Yaskawa INFORM job: u_tourne2TRJ1.JBI

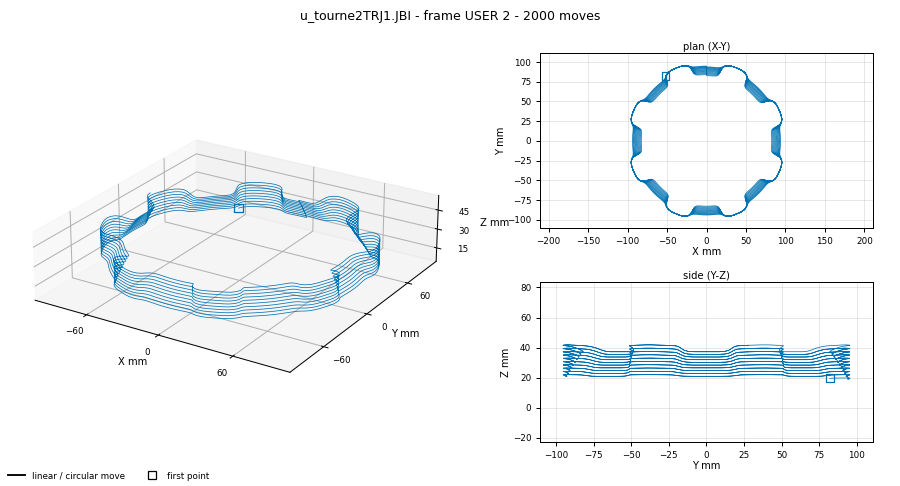
[picture p0: tool path of u_tourne2TRJ1.JBI in frame USER 2, 2000 of 2000 moves have a stored position in this frame; points joined in program order, loops and branches not executed]
/JOB
//NAME u_tourne2TRJ1
///FOLDERNAME DEMO
//POS
///NPOS 2000,0,0,0,0,0
///USER 2
///TOOL 7
///POSTYPE USER
///RECTAN
///RCONF 1,0,0,0,0,0,0,0,0,0,0,0,0,0,0,0,0,0,0,0,0,0,0,0
C00000=-51.961,81.931,19.493,-175.4388,10.0982,0.0000
C00001=-51.163,83.502,19.627,-176.4596,6.1367,0.0000
C00002=-49.917,85.194,19.692,-177.1700,3.1394,0.0000
C00003=-47.874,87.106,19.726,-178.6245,1.1234,0.0000
C00004=-45.272,88.975,19.753,-179.7708,0.1490,0.0000
C00005=-42.449,90.515,19.780,-179.9312,0.0344,0.0000
C00006=-39.659,91.796,19.798,-179.9943,0.0057,0.0000
C00007=-36.867,92.953,19.798,-179.9943,0.0057,0.0000
C00008=-33.988,94.020,19.780,-179.9255,0.0229,0.0000
C00009=-30.903,94.927,19.753,-179.7307,0.0630,0.0000
C00010=-27.741,95.446,19.726,-178.2350,0.1777,0.0000
C00011=-24.945,95.538,19.692,-175.7793,-0.2183,0.0000
C00012=-22.867,95.222,19.627,-173.1679,-1.8469,0.0000
C00013=-21.192,94.676,19.493,-169.6643,-3.9748,0.0000
C00014=-19.540,94.146,19.309,-163.8596,-4.8117,0.0000
C00015=-17.528,93.824,19.120,-157.6161,-2.4729,0.0000
C00016=-14.592,93.857,18.976,-154.0604,1.6120,0.0000
C00017=-10.190,94.262,18.917,-153.0810,2.7315,0.0000
C00018=-5.317,94.652,18.914,-152.9505,1.6728,0.0000
C00019=0.000,94.804,18.916,-152.9225,0.0000,0.0000
C00020=0.000,93.772,20.859,-151.1719,0.0000,0.0000
C00021=5.223,93.624,20.857,-151.1993,-1.7981,0.0000
C00022=10.031,93.243,20.860,-151.3314,-2.8344,0.0000
C00023=14.399,92.874,20.935,-152.4021,-1.1056,0.0000
C00024=17.292,92.935,21.118,-156.8218,4.1655,0.0000
C00025=19.271,93.399,21.361,-164.4290,6.3625,0.0000
C00026=20.902,94.108,21.598,-170.7324,4.7887,0.0000
C00027=22.556,94.852,21.773,-173.9796,2.3281,0.0000
C00028=24.607,95.353,21.858,-176.1467,0.4709,0.0000
C00029=27.423,95.407,21.902,-178.4241,-0.0974,0.0000
C00030=30.651,94.973,21.938,-179.8453,-0.0344,0.0000
C00031=33.828,94.073,21.973,-179.9370,-0.0229,0.0000
C00032=36.813,92.974,21.997,-179.9943,-0.0000,0.0000
C00033=39.712,91.773,21.997,-179.9943,-0.0057,0.0000
C00034=42.599,90.440,21.973,-179.9370,-0.0286,0.0000
C00035=45.483,88.829,21.938,-179.8682,-0.0859,0.0000
C00036=48.072,86.854,21.902,-178.8194,-1.0431,0.0000
C00037=50.025,84.825,21.858,-177.6067,-3.0580,0.0000
C00038=51.121,83.020,21.773,-177.3726,-5.9006,0.0000
C00039=51.765,81.324,21.598,-176.7879,-9.9076,0.0000
C00040=52.416,79.670,21.361,-173.2596,-15.4266,0.0000
C00041=53.488,77.942,21.118,-165.8932,-19.5057,0.0000
C00042=55.491,75.854,20.935,-159.0305,-19.5985,0.0000
C00043=58.840,73.026,20.860,-157.1383,-19.3709,0.0000
C00044=62.509,69.895,20.857,-157.6594,-20.1305,0.0000
C00045=66.307,66.307,20.859,-158.7328,-21.2672,0.0000
C00046=69.895,62.509,20.857,-159.8695,-22.3406,0.0000
C00047=73.026,58.840,20.860,-160.6291,-22.8617,0.0000
C00048=75.854,55.491,20.935,-160.4015,-20.9695,0.0000
C00049=77.942,53.488,21.118,-160.4943,-14.1068,0.0000
C00050=79.670,52.416,21.361,-164.5734,-6.7404,0.0000
C00051=81.324,51.765,21.598,-170.0924,-3.2121,0.0000
C00052=83.020,51.121,21.773,-174.0994,-2.6274,0.0000
C00053=84.825,50.025,21.858,-176.9420,-2.3933,0.0000
C00054=86.854,48.072,21.902,-178.9569,-1.1806,0.0000
C00055=88.829,45.483,21.938,-179.9141,-0.1318,0.0000
C00056=90.440,42.599,21.973,-179.9714,-0.0630,0.0000
C00057=91.773,39.712,21.997,-179.9943,-0.0057,0.0000
C00058=92.974,36.813,21.997,-180.0000,-0.0057,0.0000
C00059=94.073,33.828,21.973,-179.9771,-0.0630,0.0000
C00060=94.973,30.651,21.938,-179.9656,-0.1547,0.0000
C00061=95.407,27.423,21.902,-179.9026,-1.5759,0.0000
C00062=95.353,24.607,21.858,179.5291,-3.8533,0.0000
C00063=94.852,22.556,21.773,177.6719,-6.0204,0.0000
C00064=94.108,20.902,21.598,175.2113,-9.2676,0.0000
C00065=93.399,19.271,21.361,173.6375,-15.5710,0.0000
C00066=92.935,17.292,21.118,175.8345,-23.1782,0.0000
C00067=92.874,14.399,20.935,-178.8944,-27.5979,0.0000
C00068=93.243,10.031,20.860,-177.1656,-28.6686,0.0000
C00069=93.624,5.223,20.857,-178.2019,-28.8007,0.0000
C00070=93.772,0.000,20.859,180.0000,-28.8281,0.0000
C00071=93.624,-5.223,20.857,178.2019,-28.8007,0.0000
C00072=93.243,-10.031,20.860,177.1656,-28.6686,0.0000
C00073=92.875,-14.399,20.935,178.8944,-27.5979,0.0000
C00074=92.935,-17.292,21.118,-175.8345,-23.1782,0.0000
C00075=93.399,-19.271,21.361,-173.6375,-15.5710,0.0000
C00076=94.108,-20.902,21.598,-175.2113,-9.2676,0.0000
C00077=94.852,-22.556,21.773,-177.6719,-6.0204,0.0000
C00078=95.353,-24.607,21.858,-179.5291,-3.8533,0.0000
C00079=95.407,-27.423,21.902,179.9026,-1.5759,0.0000
C00080=94.973,-30.651,21.938,179.9656,-0.1547,0.0000
C00081=94.073,-33.828,21.973,179.9771,-0.0630,0.0000
C00082=92.974,-36.813,21.997,180.0000,-0.0057,0.0000
C00083=91.773,-39.712,21.997,179.9943,-0.0057,0.0000
C00084=90.440,-42.599,21.973,179.9714,-0.0630,0.0000
C00085=88.829,-45.483,21.938,179.9141,-0.1318,0.0000
C00086=86.854,-48.072,21.902,178.9569,-1.1806,0.0000
C00087=84.825,-50.025,21.858,176.9420,-2.3933,0.0000
C00088=83.020,-51.121,21.773,174.0994,-2.6274,0.0000
C00089=81.324,-51.765,21.598,170.0924,-3.2121,0.0000
C00090=79.670,-52.416,21.361,164.5734,-6.7404,0.0000
C00091=77.942,-53.488,21.118,160.4943,-14.1068,0.0000
C00092=75.854,-55.491,20.935,160.4015,-20.9695,0.0000
C00093=73.026,-58.840,20.860,160.6291,-22.8617,0.0000
C00094=69.895,-62.509,20.857,159.8695,-22.3406,0.0000
C00095=66.307,-66.307,20.859,158.7328,-21.2672,0.0000
C00096=62.509,-69.895,20.857,157.6594,-20.1305,0.0000
C00097=58.840,-73.026,20.860,157.1383,-19.3709,0.0000
C00098=55.491,-75.854,20.935,159.0305,-19.5985,0.0000
C00099=53.488,-77.942,21.118,165.8932,-19.5057,0.0000
C00100=52.416,-79.670,21.361,173.2596,-15.4266,0.0000
C00101=51.765,-81.324,21.598,176.7879,-9.9076,0.0000
C00102=51.121,-83.020,21.773,177.3726,-5.9006,0.0000
C00103=50.025,-84.825,21.858,177.6067,-3.0580,0.0000
C00104=48.072,-86.854,21.902,178.8194,-1.0431,0.0000
C00105=45.483,-88.829,21.938,179.8682,-0.0859,0.0000
C00106=42.599,-90.440,21.973,179.9370,-0.0286,0.0000
C00107=39.712,-91.773,21.997,179.9943,-0.0057,0.0000
C00108=36.813,-92.974,21.997,179.9943,-0.0000,0.0000
C00109=33.828,-94.073,21.973,179.9370,-0.0229,0.0000
C00110=30.651,-94.973,21.938,179.8453,-0.0344,0.0000
C00111=27.423,-95.407,21.902,178.4241,-0.0974,0.0000
C00112=24.607,-95.353,21.858,176.1467,0.4709,0.0000
C00113=22.556,-94.852,21.773,173.9796,2.3281,0.0000
C00114=20.902,-94.108,21.598,170.7324,4.7887,0.0000
C00115=19.271,-93.399,21.361,164.4290,6.3625,0.0000
C00116=17.292,-92.935,21.118,156.8218,4.1655,0.0000
C00117=14.399,-92.874,20.935,152.4021,-1.1056,0.0000
C00118=10.031,-93.243,20.860,151.3314,-2.8344,0.0000
C00119=5.223,-93.624,20.857,151.1993,-1.7981,0.0000
C00120=0.000,-93.772,20.859,151.1719,0.0000,0.0000
C00121=0.000,-93.772,20.859,151.1719,0.0000,0.0000
C00122=-5.223,-93.624,20.857,151.1993,1.7981,0.0000
C00123=-10.031,-93.243,20.860,151.3314,2.8344,0.0000
C00124=-14.399,-92.875,20.935,152.4021,1.1056,0.0000
C00125=-17.292,-92.935,21.118,156.8218,-4.1655,0.0000
C00126=-19.271,-93.399,21.361,164.4290,-6.3625,0.0000
C00127=-20.902,-94.108,21.598,170.7324,-4.7887,0.0000
C00128=-22.556,-94.852,21.773,173.9796,-2.3281,0.0000
C00129=-24.607,-95.353,21.858,176.1467,-0.4709,0.0000
C00130=-27.423,-95.407,21.902,178.4241,0.0974,0.0000
C00131=-30.651,-94.973,21.938,179.8453,0.0344,0.0000
C00132=-33.828,-94.073,21.973,179.9370,0.0229,0.0000
C00133=-36.813,-92.974,21.997,179.9943,0.0000,0.0000
C00134=-39.712,-91.773,21.997,179.9943,0.0057,0.0000
C00135=-42.599,-90.440,21.973,179.9370,0.0286,0.0000
C00136=-45.483,-88.829,21.938,179.8682,0.0859,0.0000
C00137=-48.072,-86.854,21.902,178.8194,1.0431,0.0000
C00138=-50.025,-84.825,21.858,177.6067,3.0580,0.0000
C00139=-51.121,-83.020,21.773,177.3726,5.9006,0.0000
C00140=-51.765,-81.324,21.598,176.7879,9.9076,0.0000
C00141=-52.416,-79.670,21.361,173.2596,15.4266,0.0000
C00142=-53.488,-77.942,21.118,165.8932,19.5057,0.0000
C00143=-55.491,-75.854,20.935,159.0305,19.5985,0.0000
C00144=-58.840,-73.026,20.860,157.1383,19.3709,0.0000
C00145=-62.509,-69.895,20.857,157.6594,20.1305,0.0000
C00146=-66.307,-66.307,20.859,158.7328,21.2672,0.0000
C00147=-69.895,-62.509,20.857,159.8695,22.3406,0.0000
C00148=-73.026,-58.840,20.860,160.6291,22.8617,0.0000
C00149=-75.854,-55.491,20.935,160.4015,20.9695,0.0000
C00150=-77.942,-53.488,21.118,160.4943,14.1068,0.0000
C00151=-79.670,-52.416,21.361,164.5734,6.7404,0.0000
C00152=-81.324,-51.765,21.598,170.0924,3.2121,0.0000
C00153=-83.020,-51.121,21.773,174.0994,2.6274,0.0000
C00154=-84.825,-50.025,21.858,176.9420,2.3933,0.0000
C00155=-86.854,-48.072,21.902,178.9569,1.1806,0.0000
C00156=-88.829,-45.483,21.938,179.9141,0.1318,0.0000
C00157=-90.440,-42.599,21.973,179.9714,0.0630,0.0000
C00158=-91.773,-39.712,21.997,179.9943,0.0057,0.0000
C00159=-92.974,-36.813,21.997,180.0000,0.0057,0.0000
C00160=-94.073,-33.828,21.973,179.9771,0.0630,0.0000
C00161=-94.973,-30.651,21.938,179.9656,0.1547,0.0000
C00162=-95.407,-27.423,21.902,179.9026,1.5759,0.0000
C00163=-95.353,-24.607,21.858,-179.5291,3.8533,0.0000
C00164=-94.852,-22.556,21.773,-177.6719,6.0204,0.0000
C00165=-94.108,-20.902,21.598,-175.2113,9.2676,0.0000
C00166=-93.399,-19.271,21.361,-173.6375,15.5710,0.0000
C00167=-92.935,-17.292,21.118,-175.8345,23.1782,0.0000
C00168=-92.874,-14.399,20.935,178.8944,27.5979,0.0000
C00169=-93.243,-10.031,20.860,177.1656,28.6686,0.0000
C00170=-93.624,-5.223,20.857,178.2019,28.8007,0.0000
C00171=-93.772,0.000,20.859,-180.0000,28.8281,0.0000
C00172=-93.624,5.223,20.857,-178.2019,28.8007,0.0000
C00173=-93.243,10.031,20.860,-177.1656,28.6686,0.0000
C00174=-92.875,14.399,20.935,-178.8944,27.5979,0.0000
C00175=-92.935,17.292,21.118,175.8345,23.1782,0.0000
C00176=-93.399,19.271,21.361,173.6375,15.5710,0.0000
C00177=-94.108,20.902,21.598,175.2113,9.2676,0.0000
C00178=-94.852,22.556,21.773,177.6719,6.0204,0.0000
C00179=-95.353,24.607,21.858,179.5291,3.8533,0.0000
C00180=-95.407,27.423,21.902,-179.9026,1.5759,0.0000
C00181=-94.973,30.651,21.938,-179.9656,0.1547,0.0000
C00182=-94.073,33.828,21.973,-179.9771,0.0630,0.0000
C00183=-92.974,36.813,21.997,-180.0000,0.0057,0.0000
C00184=-91.773,39.712,21.997,-179.9943,0.0057,0.0000
C00185=-90.440,42.599,21.973,-179.9714,0.0630,0.0000
C00186=-88.829,45.483,21.938,-179.9141,0.1318,0.0000
C00187=-86.854,48.072,21.902,-178.9569,1.1806,0.0000
C00188=-84.825,50.025,21.858,-176.9420,2.3933,0.0000
C00189=-83.020,51.121,21.773,-174.0994,2.6274,0.0000
C00190=-81.324,51.765,21.598,-170.0924,3.2121,0.0000
C00191=-79.670,52.416,21.361,-164.5734,6.7404,0.0000
C00192=-77.942,53.488,21.118,-160.4943,14.1068,0.0000
C00193=-75.854,55.491,20.935,-160.4015,20.9695,0.0000
C00194=-73.026,58.840,20.860,-160.6291,22.8617,0.0000
C00195=-69.895,62.509,20.857,-159.8695,22.3406,0.0000
C00196=-66.307,66.307,20.859,-158.7328,21.2672,0.0000
C00197=-62.509,69.895,20.857,-157.6594,20.1305,0.0000
C00198=-58.840,73.026,20.860,-157.1383,19.3709,0.0000
C00199=-55.491,75.854,20.935,-159.0305,19.5985,0.0000
C00200=-53.488,77.942,21.118,-165.8932,19.5057,0.0000
C00201=-52.416,79.670,21.361,-173.2596,15.4266,0.0000
C00202=-51.765,81.324,21.598,-176.7879,9.9076,0.0000
C00203=-51.121,83.020,21.773,-177.3726,5.9006,0.0000
C00204=-50.025,84.825,21.858,-177.6067,3.0580,0.0000
C00205=-48.072,86.854,21.902,-178.8194,1.0431,0.0000
C00206=-45.483,88.829,21.938,-179.8682,0.0859,0.0000
C00207=-42.599,90.440,21.973,-179.9370,0.0286,0.0000
C00208=-39.712,91.773,21.997,-179.9943,0.0057,0.0000
C00209=-36.813,92.974,21.997,-179.9943,0.0000,0.0000
C00210=-33.828,94.073,21.973,-179.9370,0.0229,0.0000
C00211=-30.651,94.973,21.938,-179.8453,0.0344,0.0000
C00212=-27.423,95.407,21.902,-178.4241,0.0974,0.0000
C00213=-24.607,95.353,21.858,-176.1467,-0.4709,0.0000
C00214=-22.556,94.852,21.773,-173.9796,-2.3281,0.0000
C00215=-20.902,94.108,21.598,-170.7324,-4.7887,0.0000
C00216=-19.271,93.399,21.361,-164.4290,-6.3625,0.0000
C00217=-17.292,92.935,21.118,-156.8218,-4.1655,0.0000
C00218=-14.399,92.875,20.935,-152.4021,1.1056,0.0000
C00219=-10.031,93.243,20.860,-151.3314,2.8344,0.0000
C00220=-5.223,93.624,20.857,-151.1993,1.7981,0.0000
C00221=0.000,93.772,20.859,-151.1719,0.0000,0.0000
C00222=0.000,92.684,22.771,-149.6091,0.0000,0.0000
C00223=5.124,92.540,22.769,-149.6408,-1.9058,0.0000
C00224=9.864,92.169,22.773,-149.7749,-2.8915,0.0000
C00225=14.194,91.838,22.865,-150.9615,-0.4587,0.0000
C00226=17.042,91.994,23.091,-156.4945,5.9914,0.0000
C00227=18.986,92.606,23.393,-165.5238,7.6283,0.0000
C00228=20.592,93.503,23.691,-172.1229,5.1950,0.0000
C00229=22.223,94.456,23.912,-175.0616,2.5313,0.0000
C00230=24.245,95.156,24.019,-176.7035,0.6543,0.0000
C00231=27.082,95.366,24.075,-178.6935,-0.0287,0.0000
C00232=30.380,95.022,24.120,-179.9771,-0.0057,0.0000
C00233=33.658,94.129,24.166,-179.9427,-0.0172,0.0000
C00234=36.755,92.996,24.196,-179.9943,-0.0000,0.0000
C00235=39.769,91.748,24.196,-179.9943,-0.0000,0.0000
C00236=42.760,90.359,24.166,-179.9484,-0.0229,0.0000
C00237=45.709,88.673,24.120,-179.9828,-0.0115,0.0000
C00238=48.284,86.584,24.075,-179.0544,-0.9055,0.0000
C00239=50.142,84.429,24.019,-178.1296,-2.7928,0.0000
C00240=51.076,82.504,23.912,-178.2908,-5.2754,0.0000
C00241=51.556,80.678,23.691,-178.0785,-9.2060,0.0000
C00242=52.057,78.907,23.393,-174.9767,-15.4952,0.0000
C00243=52.999,77.101,23.091,-166.8652,-20.8965,0.0000
C00244=54.903,74.976,22.865,-158.2902,-21.1534,0.0000
C00245=58.198,72.148,22.773,-155.8794,-20.6200,0.0000
C00246=61.813,69.059,22.769,-156.3563,-21.3360,0.0000
C00247=65.538,65.538,22.771,-157.4774,-22.5226,0.0000
C00248=69.059,61.813,22.769,-158.6640,-23.6437,0.0000
C00249=72.148,58.198,22.773,-159.3800,-24.1206,0.0000
C00250=74.976,54.903,22.865,-158.8466,-21.7155,0.0000
C00251=77.101,52.999,23.091,-159.1035,-13.1348,0.0000
C00252=78.907,52.057,23.393,-164.5048,-5.0233,0.0000
C00253=80.678,51.556,23.691,-170.7940,-1.9215,0.0000
C00254=82.504,51.076,23.912,-174.7246,-1.7092,0.0000
C00255=84.429,50.142,24.019,-177.2072,-1.8704,0.0000
C00256=86.584,48.284,24.075,-179.0945,-0.9456,0.0000
C00257=88.673,45.709,24.120,-179.9885,-0.0172,0.0000
C00258=90.359,42.760,24.166,-179.9771,-0.0516,0.0000
C00259=91.748,39.769,24.196,-180.0000,-0.0057,0.0000
C00260=92.996,36.755,24.196,-180.0000,-0.0057,0.0000
C00261=94.129,33.658,24.166,-179.9828,-0.0573,0.0000
C00262=95.022,30.380,24.120,-179.9943,-0.0229,0.0000
C00263=95.366,27.082,24.075,-179.9713,-1.3065,0.0000
C00264=95.156,24.245,24.019,179.3457,-3.2965,0.0000
C00265=94.456,22.223,23.912,177.4687,-4.9384,0.0000
C00266=93.503,20.592,23.691,174.8050,-7.8771,0.0000
C00267=92.606,18.986,23.393,172.3717,-14.4762,0.0000
C00268=91.994,17.042,23.091,174.0086,-23.5055,0.0000
C00269=91.838,14.194,22.865,-179.5413,-29.0385,0.0000
C00270=92.169,9.864,22.773,-177.1085,-30.2251,0.0000
C00271=92.540,5.124,22.769,-178.0942,-30.3592,0.0000
C00272=92.684,0.000,22.771,180.0000,-30.3909,0.0000
C00273=92.540,-5.124,22.769,178.0942,-30.3592,0.0000
C00274=92.169,-9.864,22.773,177.1085,-30.2251,0.0000
C00275=91.838,-14.194,22.865,179.5413,-29.0385,0.0000
C00276=91.994,-17.042,23.091,-174.0086,-23.5055,0.0000
C00277=92.606,-18.986,23.393,-172.3717,-14.4762,0.0000
C00278=93.503,-20.592,23.691,-174.8050,-7.8771,0.0000
C00279=94.456,-22.223,23.912,-177.4687,-4.9384,0.0000
C00280=95.156,-24.245,24.019,-179.3457,-3.2965,0.0000
C00281=95.366,-27.082,24.075,179.9713,-1.3065,0.0000
C00282=95.022,-30.380,24.120,179.9943,-0.0229,0.0000
C00283=94.129,-33.658,24.166,179.9828,-0.0573,0.0000
C00284=92.996,-36.755,24.196,180.0000,-0.0057,0.0000
C00285=91.748,-39.769,24.196,180.0000,-0.0057,0.0000
C00286=90.359,-42.760,24.166,179.9771,-0.0516,0.0000
C00287=88.673,-45.709,24.120,179.9885,-0.0172,0.0000
C00288=86.584,-48.284,24.075,179.0945,-0.9456,0.0000
C00289=84.429,-50.142,24.019,177.2072,-1.8704,0.0000
C00290=82.504,-51.076,23.912,174.7246,-1.7092,0.0000
C00291=80.678,-51.556,23.691,170.7940,-1.9215,0.0000
C00292=78.907,-52.057,23.393,164.5048,-5.0233,0.0000
C00293=77.101,-52.999,23.091,159.1035,-13.1348,0.0000
C00294=74.976,-54.903,22.865,158.8466,-21.7098,0.0000
C00295=72.148,-58.198,22.773,159.3800,-24.1206,0.0000
C00296=69.059,-61.813,22.769,158.6640,-23.6437,0.0000
C00297=65.538,-65.538,22.771,157.4774,-22.5226,0.0000
C00298=61.813,-69.059,22.769,156.3563,-21.3360,0.0000
C00299=58.198,-72.148,22.773,155.8794,-20.6200,0.0000
C00300=54.903,-74.976,22.865,158.2845,-21.1534,0.0000
C00301=52.999,-77.101,23.091,166.8652,-20.8965,0.0000
C00302=52.057,-78.907,23.393,174.9767,-15.4952,0.0000
C00303=51.556,-80.678,23.691,178.0785,-9.2060,0.0000
C00304=51.076,-82.504,23.912,178.2908,-5.2754,0.0000
C00305=50.142,-84.429,24.019,178.1296,-2.7928,0.0000
C00306=48.284,-86.584,24.075,179.0544,-0.9055,0.0000
C00307=45.709,-88.673,24.120,179.9828,-0.0115,0.0000
C00308=42.760,-90.359,24.166,179.9484,-0.0229,0.0000
C00309=39.769,-91.748,24.196,179.9943,-0.0000,0.0000
C00310=36.755,-92.996,24.196,179.9943,-0.0000,0.0000
C00311=33.658,-94.129,24.166,179.9427,-0.0172,0.0000
C00312=30.380,-95.022,24.120,179.9771,-0.0057,0.0000
C00313=27.082,-95.366,24.075,178.6935,-0.0287,0.0000
C00314=24.245,-95.156,24.019,176.7035,0.6543,0.0000
C00315=22.223,-94.456,23.912,175.0616,2.5313,0.0000
C00316=20.592,-93.503,23.691,172.1229,5.1950,0.0000
C00317=18.986,-92.606,23.393,165.5238,7.6283,0.0000
C00318=17.042,-91.994,23.091,156.4945,5.9914,0.0000
C00319=14.194,-91.838,22.865,150.9615,-0.4587,0.0000
C00320=9.864,-92.169,22.773,149.7749,-2.8915,0.0000
C00321=5.124,-92.540,22.769,149.6408,-1.9058,0.0000
C00322=0.000,-92.684,22.771,149.6091,0.0000,0.0000
C00323=0.000,-92.684,22.771,149.6091,0.0000,0.0000
C00324=-5.124,-92.540,22.769,149.6408,1.9058,0.0000
C00325=-9.864,-92.169,22.773,149.7749,2.8915,0.0000
C00326=-14.194,-91.838,22.865,150.9615,0.4587,0.0000
C00327=-17.042,-91.994,23.091,156.4945,-5.9914,0.0000
C00328=-18.986,-92.606,23.393,165.5238,-7.6283,0.0000
C00329=-20.592,-93.503,23.691,172.1229,-5.1950,0.0000
C00330=-22.223,-94.456,23.912,175.0616,-2.5313,0.0000
C00331=-24.245,-95.156,24.019,176.7035,-0.6543,0.0000
C00332=-27.082,-95.366,24.075,178.6935,0.0287,0.0000
C00333=-30.380,-95.022,24.120,179.9771,0.0057,0.0000
C00334=-33.658,-94.129,24.166,179.9427,0.0172,0.0000
C00335=-36.755,-92.996,24.196,179.9943,0.0000,0.0000
C00336=-39.769,-91.748,24.196,179.9943,0.0000,0.0000
C00337=-42.760,-90.359,24.166,179.9484,0.0229,0.0000
C00338=-45.709,-88.673,24.120,179.9828,0.0115,0.0000
C00339=-48.284,-86.584,24.075,179.0544,0.9055,0.0000
C00340=-50.142,-84.429,24.019,178.1296,2.7928,0.0000
C00341=-51.076,-82.504,23.912,178.2908,5.2754,0.0000
C00342=-51.556,-80.678,23.691,178.0785,9.2060,0.0000
C00343=-52.057,-78.907,23.393,174.9767,15.4952,0.0000
C00344=-52.999,-77.101,23.091,166.8652,20.8965,0.0000
C00345=-54.903,-74.976,22.865,158.2902,21.1534,0.0000
C00346=-58.198,-72.148,22.773,155.8794,20.6200,0.0000
C00347=-61.813,-69.059,22.769,156.3563,21.3360,0.0000
C00348=-65.538,-65.538,22.771,157.4774,22.5226,0.0000
C00349=-69.059,-61.813,22.769,158.6640,23.6437,0.0000
C00350=-72.148,-58.198,22.773,159.3800,24.1206,0.0000
C00351=-74.976,-54.903,22.865,158.8466,21.7155,0.0000
C00352=-77.101,-52.999,23.091,159.1035,13.1348,0.0000
C00353=-78.907,-52.057,23.393,164.5048,5.0233,0.0000
C00354=-80.678,-51.556,23.691,170.7940,1.9215,0.0000
C00355=-82.504,-51.076,23.912,174.7246,1.7092,0.0000
C00356=-84.429,-50.142,24.019,177.2072,1.8704,0.0000
C00357=-86.584,-48.284,24.075,179.0945,0.9456,0.0000
C00358=-88.673,-45.709,24.120,179.9885,0.0172,0.0000
C00359=-90.359,-42.760,24.166,179.9771,0.0516,0.0000
C00360=-91.748,-39.769,24.196,180.0000,0.0057,0.0000
C00361=-92.996,-36.755,24.196,180.0000,0.0057,0.0000
C00362=-94.129,-33.658,24.166,179.9828,0.0573,0.0000
C00363=-95.022,-30.380,24.120,179.9943,0.0229,0.0000
C00364=-95.366,-27.082,24.075,179.9713,1.3065,0.0000
C00365=-95.156,-24.245,24.019,-179.3457,3.2965,0.0000
C00366=-94.456,-22.223,23.912,-177.4687,4.9384,0.0000
C00367=-93.503,-20.592,23.691,-174.8050,7.8771,0.0000
C00368=-92.606,-18.986,23.393,-172.3717,14.4762,0.0000
C00369=-91.994,-17.042,23.091,-174.0086,23.5055,0.0000
C00370=-91.838,-14.194,22.865,179.5413,29.0385,0.0000
C00371=-92.169,-9.864,22.773,177.1085,30.2251,0.0000
C00372=-92.540,-5.124,22.769,178.0942,30.3592,0.0000
C00373=-92.684,0.000,22.771,-180.0000,30.3909,0.0000
C00374=-92.540,5.124,22.769,-178.0942,30.3592,0.0000
C00375=-92.169,9.864,22.773,-177.1085,30.2251,0.0000
C00376=-91.838,14.194,22.865,-179.5413,29.0385,0.0000
C00377=-91.994,17.042,23.091,174.0086,23.5055,0.0000
C00378=-92.606,18.986,23.393,172.3717,14.4762,0.0000
C00379=-93.503,20.592,23.691,174.8050,7.8771,0.0000
C00380=-94.456,22.223,23.912,177.4687,4.9384,0.0000
C00381=-95.156,24.245,24.019,179.3457,3.2965,0.0000
C00382=-95.366,27.082,24.075,-179.9713,1.3065,0.0000
C00383=-95.022,30.380,24.120,-179.9943,0.0229,0.0000
C00384=-94.129,33.658,24.166,-179.9828,0.0573,0.0000
C00385=-92.996,36.755,24.196,-180.0000,0.0057,0.0000
C00386=-91.748,39.769,24.196,-180.0000,0.0057,0.0000
C00387=-90.359,42.760,24.166,-179.9771,0.0516,0.0000
C00388=-88.673,45.709,24.120,-179.9885,0.0172,0.0000
C00389=-86.584,48.284,24.075,-179.0945,0.9456,0.0000
C00390=-84.429,50.142,24.019,-177.2072,1.8704,0.0000
C00391=-82.504,51.076,23.912,-174.7246,1.7092,0.0000
C00392=-80.678,51.556,23.691,-170.7940,1.9215,0.0000
C00393=-78.907,52.057,23.393,-164.5048,5.0233,0.0000
C00394=-77.101,52.999,23.091,-159.1035,13.1348,0.0000
C00395=-74.976,54.903,22.865,-158.8466,21.7098,0.0000
C00396=-72.148,58.198,22.773,-159.3800,24.1206,0.0000
C00397=-69.059,61.813,22.769,-158.6640,23.6437,0.0000
C00398=-65.538,65.538,22.771,-157.4774,22.5226,0.0000
C00399=-61.813,69.059,22.769,-156.3563,21.3360,0.0000
C00400=-58.198,72.148,22.773,-155.8794,20.6200,0.0000
C00401=-54.903,74.976,22.865,-158.2845,21.1534,0.0000
C00402=-52.999,77.101,23.091,-166.8652,20.8965,0.0000
C00403=-52.057,78.907,23.393,-174.9767,15.4952,0.0000
C00404=-51.556,80.678,23.691,-178.0785,9.2060,0.0000
C00405=-51.076,82.504,23.912,-178.2908,5.2754,0.0000
C00406=-50.142,84.429,24.019,-178.1296,2.7928,0.0000
C00407=-48.284,86.584,24.075,-179.0544,0.9055,0.0000
C00408=-45.709,88.673,24.120,-179.9828,0.0115,0.0000
C00409=-42.760,90.359,24.166,-179.9484,0.0229,0.0000
C00410=-39.769,91.748,24.196,-179.9943,0.0000,0.0000
C00411=-36.755,92.996,24.196,-179.9943,0.0000,0.0000
C00412=-33.658,94.129,24.166,-179.9427,0.0172,0.0000
C00413=-30.380,95.022,24.120,-179.9771,0.0057,0.0000
C00414=-27.082,95.366,24.075,-178.6935,0.0287,0.0000
C00415=-24.245,95.156,24.019,-176.7035,-0.6543,0.0000
C00416=-22.223,94.456,23.912,-175.0616,-2.5313,0.0000
C00417=-20.592,93.503,23.691,-172.1229,-5.1950,0.0000
C00418=-18.986,92.606,23.393,-165.5238,-7.6283,0.0000
C00419=-17.042,91.994,23.091,-156.4945,-5.9914,0.0000
C00420=-14.194,91.838,22.865,-150.9615,0.4587,0.0000
C00421=-9.864,92.169,22.773,-149.7749,2.8915,0.0000
C00422=-5.124,92.540,22.769,-149.6408,1.9058,0.0000
C00423=0.000,92.684,22.771,-149.6091,0.0000,0.0000
C00424=0.000,91.548,24.655,-148.2236,0.0000,0.0000
C00425=5.020,91.408,24.652,-148.2498,-2.0079,0.0000
C00426=9.690,91.047,24.657,-148.3861,-2.9135,0.0000
C00427=13.981,90.755,24.767,-149.7221,0.3185,0.0000
C00428=16.781,91.008,25.041,-156.6444,7.8331,0.0000
C00429=18.686,91.772,25.406,-167.0184,8.4700,0.0000
C00430=20.265,92.865,25.771,-173.6420,5.1605,0.0000
C00431=21.871,94.037,26.043,-176.2870,2.4065,0.0000
C00432=23.861,94.948,26.175,-177.4320,0.7169,0.0000
C00433=26.720,95.323,26.245,-179.0317,0.0229,0.0000
C00434=30.093,95.074,26.301,179.8682,0.0229,0.0000
C00435=33.476,94.189,26.358,-179.9599,-0.0172,0.0000
C00436=36.693,93.020,26.395,-179.9943,-0.0000,0.0000
C00437=39.829,91.721,26.395,-179.9943,-0.0000,0.0000
C00438=42.931,90.273,26.358,-179.9599,-0.0172,0.0000
C00439=45.948,88.507,26.301,179.8911,0.0802,0.0000
C00440=48.509,86.297,26.245,-179.3296,-0.6990,0.0000
C00441=50.266,84.010,26.175,-178.6924,-2.3275,0.0000
C00442=51.029,81.959,26.043,-179.0748,-4.3249,0.0000
C00443=51.336,79.995,25.771,-179.1434,-8.1179,0.0000
C00444=51.679,78.105,25.406,-176.7001,-15.0175,0.0000
C00445=52.487,76.218,25.041,-168.2468,-21.9304,0.0000
C00446=54.287,74.059,24.767,-157.7618,-22.6236,0.0000
C00447=57.528,71.231,24.657,-154.7700,-21.7654,0.0000
C00448=61.085,68.184,24.652,-155.1864,-22.4262,0.0000
C00449=64.734,64.734,24.655,-156.3434,-23.6566,0.0000
C00450=68.184,61.085,24.652,-157.5738,-24.8136,0.0000
C00451=71.231,57.528,24.657,-158.2346,-25.2300,0.0000
C00452=74.059,54.287,24.767,-157.3764,-22.2382,0.0000
C00453=76.218,52.487,25.041,-158.0696,-11.7532,0.0000
C00454=78.105,51.679,25.406,-164.9825,-3.2999,0.0000
C00455=79.995,51.336,25.771,-171.8821,-0.8566,0.0000
C00456=81.959,51.029,26.043,-175.6751,-0.9252,0.0000
C00457=84.010,50.266,26.175,-177.6725,-1.3076,0.0000
C00458=86.297,48.509,26.245,-179.3010,-0.6704,0.0000
C00459=88.507,45.948,26.301,179.9198,0.1089,0.0000
C00460=90.273,42.931,26.358,-179.9828,-0.0401,0.0000
C00461=91.721,39.829,26.395,-180.0000,-0.0057,0.0000
C00462=93.020,36.693,26.395,-180.0000,-0.0057,0.0000
C00463=94.189,33.476,26.358,-179.9828,-0.0401,0.0000
C00464=95.074,30.093,26.301,179.9771,0.1318,0.0000
C00465=95.323,26.720,26.245,179.9771,-0.9683,0.0000
C00466=94.948,23.861,26.175,179.2831,-2.5680,0.0000
C00467=94.037,21.871,26.043,177.5935,-3.7130,0.0000
C00468=92.865,20.265,25.771,174.8395,-6.3580,0.0000
C00469=91.772,18.686,25.406,171.5300,-12.9816,0.0000
C00470=91.008,16.781,25.041,172.1669,-23.3556,0.0000
C00471=90.755,13.981,24.767,179.6815,-30.2779,0.0000
C00472=91.047,9.690,24.657,-177.0865,-31.6139,0.0000
C00473=91.408,5.020,24.652,-177.9921,-31.7502,0.0000
C00474=91.548,0.000,24.655,180.0000,-31.7764,0.0000
C00475=91.408,-5.020,24.652,177.9921,-31.7502,0.0000
C00476=91.047,-9.690,24.657,177.0865,-31.6139,0.0000
C00477=90.755,-13.981,24.767,-179.6815,-30.2779,0.0000
C00478=91.008,-16.781,25.041,-172.1669,-23.3556,0.0000
C00479=91.772,-18.686,25.406,-171.5300,-12.9816,0.0000
C00480=92.865,-20.265,25.771,-174.8395,-6.3580,0.0000
C00481=94.037,-21.871,26.043,-177.5935,-3.7130,0.0000
C00482=94.948,-23.861,26.175,-179.2831,-2.5680,0.0000
C00483=95.323,-26.720,26.245,-179.9771,-0.9683,0.0000
C00484=95.074,-30.093,26.301,-179.9771,0.1318,0.0000
C00485=94.189,-33.476,26.358,179.9828,-0.0401,0.0000
C00486=93.020,-36.693,26.395,180.0000,-0.0057,0.0000
C00487=91.721,-39.829,26.395,180.0000,-0.0057,0.0000
C00488=90.273,-42.931,26.358,179.9828,-0.0401,0.0000
C00489=88.507,-45.948,26.301,-179.9198,0.1089,0.0000
C00490=86.297,-48.509,26.245,179.3010,-0.6704,0.0000
C00491=84.010,-50.266,26.175,177.6725,-1.3076,0.0000
C00492=81.959,-51.029,26.043,175.6751,-0.9252,0.0000
C00493=79.995,-51.336,25.771,171.8821,-0.8566,0.0000
C00494=78.105,-51.679,25.406,164.9825,-3.2999,0.0000
C00495=76.218,-52.487,25.041,158.0696,-11.7532,0.0000
C00496=74.059,-54.287,24.767,157.3764,-22.2382,0.0000
C00497=71.231,-57.528,24.657,158.2346,-25.2300,0.0000
C00498=68.184,-61.085,24.652,157.5738,-24.8136,0.0000
C00499=64.734,-64.734,24.655,156.3434,-23.6566,0.0000
C00500=61.085,-68.184,24.652,155.1864,-22.4262,0.0000
C00501=57.528,-71.231,24.657,154.7700,-21.7654,0.0000
C00502=54.287,-74.059,24.767,157.7618,-22.6236,0.0000
C00503=52.487,-76.218,25.041,168.2468,-21.9304,0.0000
C00504=51.679,-78.105,25.406,176.7001,-15.0175,0.0000
C00505=51.336,-79.995,25.771,179.1434,-8.1179,0.0000
C00506=51.029,-81.959,26.043,179.0748,-4.3249,0.0000
C00507=50.266,-84.010,26.175,178.6924,-2.3275,0.0000
C00508=48.509,-86.297,26.245,179.3296,-0.6990,0.0000
C00509=45.948,-88.507,26.301,-179.8911,0.0802,0.0000
C00510=42.931,-90.273,26.358,179.9599,-0.0172,0.0000
C00511=39.829,-91.721,26.395,179.9943,-0.0000,0.0000
C00512=36.693,-93.020,26.395,179.9943,-0.0000,0.0000
C00513=33.476,-94.189,26.358,179.9599,-0.0172,0.0000
C00514=30.093,-95.074,26.301,-179.8682,0.0229,0.0000
C00515=26.720,-95.323,26.245,179.0317,0.0229,0.0000
C00516=23.861,-94.948,26.175,177.4320,0.7169,0.0000
C00517=21.871,-94.037,26.043,176.2870,2.4065,0.0000
C00518=20.265,-92.865,25.771,173.6420,5.1605,0.0000
C00519=18.686,-91.772,25.406,167.0184,8.4700,0.0000
C00520=16.781,-91.008,25.041,156.6444,7.8331,0.0000
C00521=13.981,-90.755,24.767,149.7221,0.3185,0.0000
C00522=9.690,-91.047,24.657,148.3861,-2.9135,0.0000
C00523=5.020,-91.408,24.652,148.2498,-2.0079,0.0000
C00524=0.000,-91.548,24.655,148.2236,0.0000,0.0000
C00525=0.000,-91.548,24.655,148.2236,0.0000,0.0000
C00526=-5.020,-91.408,24.652,148.2498,2.0079,0.0000
C00527=-9.690,-91.047,24.657,148.3861,2.9135,0.0000
C00528=-13.981,-90.755,24.767,149.7221,-0.3185,0.0000
C00529=-16.781,-91.008,25.041,156.6444,-7.8331,0.0000
C00530=-18.686,-91.772,25.406,167.0184,-8.4700,0.0000
C00531=-20.265,-92.865,25.771,173.6420,-5.1605,0.0000
C00532=-21.871,-94.037,26.043,176.2870,-2.4065,0.0000
C00533=-23.861,-94.948,26.175,177.4320,-0.7169,0.0000
C00534=-26.720,-95.323,26.245,179.0317,-0.0229,0.0000
C00535=-30.093,-95.074,26.301,-179.8682,-0.0229,0.0000
C00536=-33.476,-94.189,26.358,179.9599,0.0172,0.0000
C00537=-36.693,-93.020,26.395,179.9943,0.0000,0.0000
C00538=-39.829,-91.721,26.395,179.9943,0.0000,0.0000
C00539=-42.931,-90.273,26.358,179.9599,0.0172,0.0000
C00540=-45.948,-88.507,26.301,-179.8911,-0.0802,0.0000
C00541=-48.509,-86.297,26.245,179.3296,0.6990,0.0000
C00542=-50.266,-84.010,26.175,178.6924,2.3275,0.0000
C00543=-51.029,-81.959,26.043,179.0748,4.3249,0.0000
C00544=-51.336,-79.995,25.771,179.1434,8.1179,0.0000
C00545=-51.679,-78.105,25.406,176.7001,15.0175,0.0000
C00546=-52.487,-76.218,25.041,168.2468,21.9304,0.0000
C00547=-54.287,-74.059,24.767,157.7618,22.6236,0.0000
C00548=-57.528,-71.231,24.657,154.7700,21.7654,0.0000
C00549=-61.085,-68.184,24.652,155.1864,22.4262,0.0000
C00550=-64.734,-64.734,24.655,156.3434,23.6566,0.0000
C00551=-68.184,-61.085,24.652,157.5738,24.8136,0.0000
C00552=-71.231,-57.528,24.657,158.2346,25.2300,0.0000
C00553=-74.059,-54.287,24.767,157.3764,22.2382,0.0000
C00554=-76.218,-52.487,25.041,158.0696,11.7532,0.0000
C00555=-78.105,-51.679,25.406,164.9825,3.2999,0.0000
C00556=-79.995,-51.336,25.771,171.8821,0.8566,0.0000
C00557=-81.959,-51.029,26.043,175.6751,0.9252,0.0000
C00558=-84.010,-50.266,26.175,177.6725,1.3076,0.0000
C00559=-86.297,-48.509,26.245,179.3010,0.6704,0.0000
C00560=-88.507,-45.948,26.301,-179.9198,-0.1089,0.0000
C00561=-90.273,-42.931,26.358,179.9828,0.0401,0.0000
C00562=-91.721,-39.829,26.395,180.0000,0.0057,0.0000
C00563=-93.020,-36.693,26.395,180.0000,0.0057,0.0000
C00564=-94.189,-33.476,26.358,179.9828,0.0401,0.0000
C00565=-95.074,-30.093,26.301,-179.9771,-0.1318,0.0000
C00566=-95.323,-26.720,26.245,-179.9771,0.9683,0.0000
C00567=-94.948,-23.861,26.175,-179.2831,2.5680,0.0000
C00568=-94.037,-21.871,26.043,-177.5935,3.7130,0.0000
C00569=-92.865,-20.265,25.771,-174.8395,6.3580,0.0000
C00570=-91.772,-18.686,25.406,-171.5300,12.9816,0.0000
C00571=-91.008,-16.781,25.041,-172.1669,23.3556,0.0000
C00572=-90.755,-13.981,24.767,-179.6815,30.2779,0.0000
C00573=-91.047,-9.690,24.657,177.0865,31.6139,0.0000
C00574=-91.408,-5.020,24.652,177.9921,31.7502,0.0000
C00575=-91.548,0.000,24.655,-180.0000,31.7764,0.0000
C00576=-91.408,5.020,24.652,-177.9921,31.7502,0.0000
C00577=-91.047,9.690,24.657,-177.0865,31.6139,0.0000
C00578=-90.755,13.981,24.767,179.6815,30.2779,0.0000
C00579=-91.008,16.781,25.041,172.1669,23.3556,0.0000
C00580=-91.772,18.686,25.406,171.5300,12.9816,0.0000
C00581=-92.865,20.265,25.771,174.8395,6.3580,0.0000
C00582=-94.037,21.871,26.043,177.5935,3.7130,0.0000
C00583=-94.948,23.861,26.175,179.2831,2.5680,0.0000
C00584=-95.323,26.720,26.245,179.9771,0.9683,0.0000
C00585=-95.074,30.093,26.301,179.9771,-0.1318,0.0000
C00586=-94.189,33.476,26.358,-179.9828,0.0401,0.0000
C00587=-93.020,36.693,26.395,-180.0000,0.0057,0.0000
C00588=-91.721,39.829,26.395,-180.0000,0.0057,0.0000
C00589=-90.273,42.931,26.358,-179.9828,0.0401,0.0000
C00590=-88.507,45.948,26.301,179.9198,-0.1089,0.0000
C00591=-86.297,48.509,26.245,-179.3010,0.6704,0.0000
C00592=-84.010,50.266,26.175,-177.6725,1.3076,0.0000
C00593=-81.959,51.029,26.043,-175.6751,0.9252,0.0000
C00594=-79.995,51.336,25.771,-171.8821,0.8566,0.0000
C00595=-78.105,51.679,25.406,-164.9825,3.2999,0.0000
C00596=-76.218,52.487,25.041,-158.0696,11.7532,0.0000
C00597=-74.059,54.287,24.767,-157.3764,22.2382,0.0000
C00598=-71.231,57.528,24.657,-158.2346,25.2300,0.0000
C00599=-68.184,61.085,24.652,-157.5738,24.8136,0.0000
C00600=-64.734,64.734,24.655,-156.3434,23.6566,0.0000
C00601=-61.085,68.184,24.652,-155.1864,22.4262,0.0000
C00602=-57.528,71.231,24.657,-154.7700,21.7654,0.0000
C00603=-54.287,74.059,24.767,-157.7618,22.6236,0.0000
C00604=-52.487,76.218,25.041,-168.2468,21.9304,0.0000
C00605=-51.679,78.105,25.406,-176.7001,15.0175,0.0000
C00606=-51.336,79.995,25.771,-179.1434,8.1179,0.0000
C00607=-51.029,81.959,26.043,-179.0748,4.3249,0.0000
C00608=-50.266,84.010,26.175,-178.6924,2.3275,0.0000
C00609=-48.509,86.297,26.245,-179.3296,0.6990,0.0000
C00610=-45.948,88.507,26.301,179.8911,-0.0802,0.0000
C00611=-42.931,90.273,26.358,-179.9599,0.0172,0.0000
C00612=-39.829,91.721,26.395,-179.9943,0.0000,0.0000
C00613=-36.693,93.020,26.395,-179.9943,0.0000,0.0000
C00614=-33.476,94.189,26.358,-179.9599,0.0172,0.0000
C00615=-30.093,95.074,26.301,179.8682,-0.0229,0.0000
C00616=-26.720,95.323,26.245,-179.0317,-0.0229,0.0000
C00617=-23.861,94.948,26.175,-177.4320,-0.7169,0.0000
C00618=-21.871,94.037,26.043,-176.2870,-2.4065,0.0000
C00619=-20.265,92.865,25.771,-173.6420,-5.1605,0.0000
C00620=-18.686,91.772,25.406,-167.0184,-8.4700,0.0000
C00621=-16.781,91.008,25.041,-156.6444,-7.8331,0.0000
C00622=-13.981,90.755,24.767,-149.7221,-0.3185,0.0000
C00623=-9.690,91.047,24.657,-148.3861,2.9135,0.0000
C00624=-5.020,91.408,24.652,-148.2498,2.0079,0.0000
C00625=0.000,91.548,24.655,-148.2236,0.0000,0.0000
C00626=0.000,90.369,26.513,-146.9901,0.0000,0.0000
C00627=4.912,90.233,26.509,-147.0206,-2.0968,0.0000
C00628=9.508,89.882,26.515,-147.1593,-2.8985,0.0000
C00629=13.759,89.629,26.645,-148.6805,1.2140,0.0000
C00630=16.509,89.983,26.968,-157.2651,9.5602,0.0000
C00631=18.373,90.901,27.402,-168.7355,8.8469,0.0000
C00632=19.923,92.196,27.838,-175.1304,4.7436,0.0000
C00633=21.502,93.597,28.166,-177.5226,1.9674,0.0000
C00634=23.458,94.728,28.327,-178.2693,0.6305,0.0000
C00635=26.340,95.277,28.411,-179.4213,0.0344,0.0000
C00636=29.791,95.129,28.479,179.6963,0.0458,0.0000
C00637=33.285,94.252,28.548,-179.9714,-0.0115,0.0000
C00638=36.628,93.045,28.594,-180.0000,-0.0000,0.0000
C00639=39.893,91.693,28.594,-180.0000,-0.0000,0.0000
C00640=43.110,90.182,28.548,-179.9714,-0.0115,0.0000
C00641=46.201,88.332,28.479,179.7536,0.1833,0.0000
C00642=48.746,85.996,28.411,-179.6161,-0.4355,0.0000
C00643=50.396,83.570,28.327,-179.2262,-1.6677,0.0000
C00644=50.979,81.387,28.166,-179.6385,-3.1414,0.0000
C00645=51.105,79.281,27.838,-179.9077,-6.7825,0.0000
C00646=51.285,77.269,27.402,-178.2394,-14.0877,0.0000
C00647=51.954,75.301,26.968,-169.9515,-22.5582,0.0000
C00648=53.649,73.106,26.645,-157.4473,-24.0017,0.0000
C00649=56.833,70.280,26.515,-153.7965,-22.8144,0.0000
C00650=60.331,67.277,26.509,-154.1417,-23.4086,0.0000
C00651=63.901,63.901,26.513,-155.3289,-24.6711,0.0000
C00652=67.277,60.331,26.509,-156.5914,-25.8583,0.0000
C00653=70.280,56.833,26.515,-157.1856,-26.2035,0.0000
C00654=73.106,53.649,26.645,-155.9983,-22.5527,0.0000
C00655=75.301,51.954,26.968,-157.4418,-10.0485,0.0000
C00656=77.269,51.285,27.402,-165.9123,-1.7606,0.0000
C00657=79.281,51.105,27.838,-173.2175,-0.0923,0.0000
C00658=81.387,50.979,28.166,-176.8586,-0.3615,0.0000
C00659=83.570,50.396,28.327,-178.3323,-0.7738,0.0000
C00660=85.996,48.746,28.411,-179.5645,-0.3839,0.0000
C00661=88.332,46.201,28.479,179.8167,0.2464,0.0000
C00662=90.182,43.110,28.548,-179.9885,-0.0286,0.0000
C00663=91.693,39.893,28.594,-180.0000,-0.0000,0.0000
C00664=93.045,36.628,28.594,-180.0000,-0.0000,0.0000
C00665=94.252,33.285,28.548,-179.9885,-0.0286,0.0000
C00666=95.129,29.791,28.479,179.9542,0.3037,0.0000
C00667=95.277,26.340,28.411,179.9656,-0.5787,0.0000
C00668=94.728,23.458,28.327,179.3695,-1.7307,0.0000
C00669=93.597,21.502,28.166,178.0326,-2.4774,0.0000
C00670=92.196,19.923,27.838,175.2564,-4.8696,0.0000
C00671=90.901,18.373,27.402,171.1531,-11.2645,0.0000
C00672=89.983,16.509,26.968,170.4398,-22.7349,0.0000
C00673=89.629,13.759,26.645,178.7860,-31.3195,0.0000
C00674=89.882,9.508,26.515,-177.1015,-32.8407,0.0000
C00675=90.233,4.912,26.509,-177.9032,-32.9794,0.0000
C00676=90.369,0.000,26.513,180.0000,-33.0099,0.0000
C00677=90.233,-4.912,26.509,177.9032,-32.9794,0.0000
C00678=89.882,-9.508,26.515,177.1015,-32.8407,0.0000
C00679=89.629,-13.759,26.645,-178.7860,-31.3195,0.0000
C00680=89.983,-16.509,26.968,-170.4398,-22.7349,0.0000
C00681=90.901,-18.373,27.402,-171.1531,-11.2645,0.0000
C00682=92.196,-19.923,27.838,-175.2564,-4.8696,0.0000
C00683=93.597,-21.502,28.166,-178.0326,-2.4774,0.0000
C00684=94.728,-23.458,28.327,-179.3695,-1.7307,0.0000
C00685=95.277,-26.340,28.411,-179.9656,-0.5787,0.0000
C00686=95.129,-29.791,28.479,-179.9542,0.3037,0.0000
C00687=94.252,-33.285,28.548,179.9885,-0.0286,0.0000
C00688=93.045,-36.628,28.594,180.0000,-0.0000,0.0000
C00689=91.693,-39.893,28.594,180.0000,-0.0000,0.0000
C00690=90.182,-43.110,28.548,179.9885,-0.0286,0.0000
C00691=88.332,-46.201,28.479,-179.8167,0.2464,0.0000
C00692=85.996,-48.746,28.411,179.5645,-0.3839,0.0000
C00693=83.570,-50.396,28.327,178.3323,-0.7738,0.0000
C00694=81.387,-50.979,28.166,176.8586,-0.3615,0.0000
C00695=79.281,-51.105,27.838,173.2175,-0.0923,0.0000
C00696=77.269,-51.285,27.402,165.9123,-1.7606,0.0000
C00697=75.301,-51.954,26.968,157.4418,-10.0485,0.0000
C00698=73.106,-53.649,26.645,155.9983,-22.5527,0.0000
C00699=70.280,-56.833,26.515,157.1856,-26.2035,0.0000
C00700=67.277,-60.331,26.509,156.5914,-25.8583,0.0000
C00701=63.901,-63.901,26.513,155.3289,-24.6711,0.0000
C00702=60.331,-67.277,26.509,154.1417,-23.4086,0.0000
C00703=56.833,-70.280,26.515,153.7965,-22.8144,0.0000
C00704=53.649,-73.106,26.645,157.4473,-24.0017,0.0000
C00705=51.954,-75.301,26.968,169.9515,-22.5582,0.0000
C00706=51.285,-77.269,27.402,178.2394,-14.0877,0.0000
C00707=51.105,-79.281,27.838,179.9077,-6.7825,0.0000
C00708=50.979,-81.387,28.166,179.6385,-3.1414,0.0000
C00709=50.396,-83.570,28.327,179.2262,-1.6677,0.0000
C00710=48.746,-85.996,28.411,179.6161,-0.4355,0.0000
C00711=46.201,-88.332,28.479,-179.7536,0.1833,0.0000
C00712=43.110,-90.182,28.548,179.9714,-0.0115,0.0000
C00713=39.893,-91.693,28.594,180.0000,-0.0000,0.0000
C00714=36.628,-93.045,28.594,180.0000,-0.0000,0.0000
C00715=33.285,-94.252,28.548,179.9714,-0.0115,0.0000
C00716=29.791,-95.129,28.479,-179.6963,0.0458,0.0000
C00717=26.340,-95.277,28.411,179.4213,0.0344,0.0000
C00718=23.458,-94.728,28.327,178.2693,0.6305,0.0000
C00719=21.502,-93.597,28.166,177.5226,1.9674,0.0000
C00720=19.923,-92.196,27.838,175.1304,4.7436,0.0000
C00721=18.373,-90.901,27.402,168.7355,8.8469,0.0000
C00722=16.509,-89.983,26.968,157.2651,9.5602,0.0000
C00723=13.759,-89.629,26.645,148.6805,1.2140,0.0000
C00724=9.508,-89.882,26.515,147.1593,-2.8985,0.0000
C00725=4.912,-90.233,26.509,147.0206,-2.0968,0.0000
C00726=0.000,-90.369,26.513,146.9901,0.0000,0.0000
C00727=0.000,-90.369,26.513,146.9901,0.0000,0.0000
C00728=-4.912,-90.233,26.509,147.0206,2.0968,0.0000
C00729=-9.508,-89.882,26.515,147.1593,2.8985,0.0000
C00730=-13.759,-89.629,26.645,148.6805,-1.2140,0.0000
C00731=-16.509,-89.983,26.968,157.2651,-9.5602,0.0000
C00732=-18.373,-90.901,27.402,168.7355,-8.8469,0.0000
C00733=-19.923,-92.196,27.838,175.1304,-4.7436,0.0000
C00734=-21.502,-93.597,28.166,177.5226,-1.9674,0.0000
C00735=-23.458,-94.728,28.327,178.2693,-0.6305,0.0000
C00736=-26.340,-95.277,28.411,179.4213,-0.0344,0.0000
C00737=-29.791,-95.129,28.479,-179.6963,-0.0458,0.0000
C00738=-33.285,-94.252,28.548,179.9714,0.0115,0.0000
C00739=-36.628,-93.045,28.594,180.0000,0.0000,0.0000
C00740=-39.893,-91.693,28.594,180.0000,0.0000,0.0000
C00741=-43.110,-90.182,28.548,179.9714,0.0115,0.0000
C00742=-46.201,-88.332,28.479,-179.7536,-0.1833,0.0000
C00743=-48.746,-85.996,28.411,179.6161,0.4355,0.0000
C00744=-50.396,-83.570,28.327,179.2262,1.6677,0.0000
C00745=-50.979,-81.387,28.166,179.6385,3.1414,0.0000
C00746=-51.105,-79.281,27.838,179.9077,6.7825,0.0000
C00747=-51.285,-77.269,27.402,178.2394,14.0877,0.0000
C00748=-51.954,-75.301,26.968,169.9515,22.5582,0.0000
C00749=-53.649,-73.106,26.645,157.4473,24.0017,0.0000
C00750=-56.833,-70.280,26.515,153.7965,22.8144,0.0000
C00751=-60.331,-67.277,26.509,154.1417,23.4086,0.0000
C00752=-63.901,-63.901,26.513,155.3289,24.6711,0.0000
C00753=-67.277,-60.331,26.509,156.5914,25.8583,0.0000
C00754=-70.280,-56.833,26.515,157.1856,26.2035,0.0000
C00755=-73.106,-53.649,26.645,155.9983,22.5527,0.0000
C00756=-75.301,-51.954,26.968,157.4418,10.0485,0.0000
C00757=-77.269,-51.285,27.402,165.9123,1.7606,0.0000
C00758=-79.281,-51.105,27.838,173.2175,0.0923,0.0000
C00759=-81.387,-50.979,28.166,176.8586,0.3615,0.0000
C00760=-83.570,-50.396,28.327,178.3323,0.7738,0.0000
C00761=-85.996,-48.746,28.411,179.5645,0.3839,0.0000
C00762=-88.332,-46.201,28.479,-179.8167,-0.2464,0.0000
C00763=-90.182,-43.110,28.548,179.9885,0.0286,0.0000
C00764=-91.693,-39.893,28.594,180.0000,0.0000,0.0000
C00765=-93.045,-36.628,28.594,180.0000,0.0000,0.0000
C00766=-94.252,-33.285,28.548,179.9885,0.0286,0.0000
C00767=-95.129,-29.791,28.479,-179.9542,-0.3037,0.0000
C00768=-95.277,-26.340,28.411,-179.9656,0.5787,0.0000
C00769=-94.728,-23.458,28.327,-179.3695,1.7307,0.0000
C00770=-93.597,-21.502,28.166,-178.0326,2.4774,0.0000
C00771=-92.196,-19.923,27.838,-175.2564,4.8696,0.0000
C00772=-90.901,-18.373,27.402,-171.1531,11.2645,0.0000
C00773=-89.983,-16.509,26.968,-170.4398,22.7349,0.0000
C00774=-89.629,-13.759,26.645,-178.7860,31.3195,0.0000
C00775=-89.882,-9.508,26.515,177.1015,32.8407,0.0000
C00776=-90.233,-4.912,26.509,177.9032,32.9794,0.0000
C00777=-90.369,0.000,26.513,-180.0000,33.0099,0.0000
C00778=-90.233,4.912,26.509,-177.9032,32.9794,0.0000
C00779=-89.882,9.508,26.515,-177.1015,32.8407,0.0000
C00780=-89.629,13.759,26.645,178.7860,31.3195,0.0000
C00781=-89.983,16.509,26.968,170.4398,22.7349,0.0000
C00782=-90.901,18.373,27.402,171.1531,11.2645,0.0000
C00783=-92.196,19.923,27.838,175.2564,4.8696,0.0000
C00784=-93.597,21.502,28.166,178.0326,2.4774,0.0000
C00785=-94.728,23.458,28.327,179.3695,1.7307,0.0000
C00786=-95.277,26.340,28.411,179.9656,0.5787,0.0000
C00787=-95.129,29.791,28.479,179.9542,-0.3037,0.0000
C00788=-94.252,33.285,28.548,-179.9885,0.0286,0.0000
C00789=-93.045,36.628,28.594,-180.0000,0.0000,0.0000
C00790=-91.693,39.893,28.594,-180.0000,0.0000,0.0000
C00791=-90.182,43.110,28.548,-179.9885,0.0286,0.0000
C00792=-88.332,46.201,28.479,179.8167,-0.2464,0.0000
C00793=-85.996,48.746,28.411,-179.5645,0.3839,0.0000
C00794=-83.570,50.396,28.327,-178.3323,0.7738,0.0000
C00795=-81.387,50.979,28.166,-176.8586,0.3615,0.0000
C00796=-79.281,51.105,27.838,-173.2175,0.0923,0.0000
C00797=-77.269,51.285,27.402,-165.9123,1.7606,0.0000
C00798=-75.301,51.954,26.968,-157.4418,10.0485,0.0000
C00799=-73.106,53.649,26.645,-155.9983,22.5527,0.0000
C00800=-70.280,56.833,26.515,-157.1856,26.2035,0.0000
C00801=-67.277,60.331,26.509,-156.5914,25.8583,0.0000
C00802=-63.901,63.901,26.513,-155.3289,24.6711,0.0000
C00803=-60.331,67.277,26.509,-154.1417,23.4086,0.0000
C00804=-56.833,70.280,26.515,-153.7965,22.8144,0.0000
C00805=-53.649,73.106,26.645,-157.4473,24.0017,0.0000
C00806=-51.954,75.301,26.968,-169.9515,22.5582,0.0000
C00807=-51.285,77.269,27.402,-178.2394,14.0877,0.0000
C00808=-51.105,79.281,27.838,-179.9077,6.7825,0.0000
C00809=-50.979,81.387,28.166,-179.6385,3.1414,0.0000
C00810=-50.396,83.570,28.327,-179.2262,1.6677,0.0000
C00811=-48.746,85.996,28.411,-179.6161,0.4355,0.0000
C00812=-46.201,88.332,28.479,179.7536,-0.1833,0.0000
C00813=-43.110,90.182,28.548,-179.9714,0.0115,0.0000
C00814=-39.893,91.693,28.594,-180.0000,0.0000,0.0000
C00815=-36.628,93.045,28.594,-180.0000,0.0000,0.0000
C00816=-33.285,94.252,28.548,-179.9714,0.0115,0.0000
C00817=-29.791,95.129,28.479,179.6963,-0.0458,0.0000
C00818=-26.340,95.277,28.411,-179.4213,-0.0344,0.0000
C00819=-23.458,94.728,28.327,-178.2693,-0.6305,0.0000
C00820=-21.502,93.597,28.166,-177.5226,-1.9674,0.0000
C00821=-19.923,92.196,27.838,-175.1304,-4.7436,0.0000
C00822=-18.373,90.901,27.402,-168.7355,-8.8469,0.0000
C00823=-16.509,89.983,26.968,-157.2651,-9.5602,0.0000
C00824=-13.759,89.629,26.645,-148.6805,-1.2140,0.0000
C00825=-9.508,89.882,26.515,-147.1593,2.8985,0.0000
C00826=-4.912,90.233,26.509,-147.0206,2.0968,0.0000
C00827=0.000,90.369,26.513,-146.9901,0.0000,0.0000
C00828=0.000,89.153,28.346,-145.9031,0.0000,0.0000
C00829=4.801,89.020,28.341,-145.9331,-2.1718,0.0000
C00830=9.321,88.681,28.348,-146.0777,-2.8448,0.0000
C00831=13.530,88.468,28.499,-147.8269,2.2135,0.0000
C00832=16.227,88.922,28.874,-158.3132,11.0590,0.0000
C00833=18.049,89.999,29.382,-170.5158,8.7912,0.0000
C00834=19.567,91.502,29.895,-176.4767,4.0390,0.0000
C00835=21.117,93.139,30.283,-178.6646,1.2724,0.0000
C00836=23.038,94.499,30.474,-179.1692,0.3782,0.0000
C00837=25.943,95.229,30.574,-179.8568,0.0172,0.0000
C00838=29.476,95.186,30.656,179.5073,0.0630,0.0000
C00839=33.085,94.318,30.738,-179.9828,-0.0057,0.0000
C00840=36.560,93.071,30.793,-180.0000,-0.0000,0.0000
C00841=39.959,91.663,30.793,-180.0000,-0.0000,0.0000
C00842=43.298,90.088,30.738,-179.9885,-0.0057,0.0000
C00843=46.464,88.150,30.656,179.6104,0.3037,0.0000
C00844=48.993,85.682,30.574,-179.9083,-0.1146,0.0000
C00845=50.531,83.111,30.474,-179.6791,-0.8537,0.0000
C00846=50.927,80.791,30.283,-179.9541,-1.8395,0.0000
C00847=50.865,78.538,29.895,179.6374,-5.3366,0.0000
C00848=50.876,76.401,29.382,-179.4947,-12.8147,0.0000
C00849=51.403,74.351,28.874,-171.8646,-22.7501,0.0000
C00850=52.989,72.123,28.499,-157.3398,-25.2777,0.0000
C00851=56.115,69.298,28.348,-152.9478,-23.7724,0.0000
C00852=59.552,66.342,28.341,-153.2084,-24.2910,0.0000
C00853=63.040,63.040,28.346,-154.4202,-25.5798,0.0000
C00854=66.342,59.552,28.341,-155.7090,-26.7916,0.0000
C00855=69.298,56.115,28.348,-156.2276,-27.0522,0.0000
C00856=72.123,52.989,28.499,-154.7223,-22.6602,0.0000
C00857=74.351,51.403,28.874,-157.2499,-8.1354,0.0000
C00858=76.401,50.876,29.382,-167.1853,-0.5053,0.0000
C00859=78.538,50.865,29.895,-174.6634,0.3626,0.0000
C00860=80.791,50.927,30.283,-178.1605,-0.0459,0.0000
C00861=83.111,50.531,30.474,-179.1463,-0.3209,0.0000
C00862=85.682,48.993,30.574,-179.8854,-0.0917,0.0000
C00863=88.150,46.464,30.656,179.6963,0.3896,0.0000
C00864=90.088,43.298,30.738,-179.9943,-0.0115,0.0000
C00865=91.663,39.959,30.793,-180.0000,-0.0000,0.0000
C00866=93.071,36.560,30.793,-180.0000,-0.0000,0.0000
C00867=94.318,33.085,30.738,-179.9943,-0.0172,0.0000
C00868=95.186,29.476,30.656,179.9370,0.4927,0.0000
C00869=95.229,25.943,30.574,179.9828,-0.1432,0.0000
C00870=94.499,23.038,30.474,179.6218,-0.8308,0.0000
C00871=93.139,21.117,30.283,178.7276,-1.3354,0.0000
C00872=91.502,19.567,29.895,175.9610,-3.5233,0.0000
C00873=89.999,18.049,29.382,171.2088,-9.4842,0.0000
C00874=88.922,16.227,28.874,168.9410,-21.6868,0.0000
C00875=88.468,13.530,28.499,177.7865,-32.1731,0.0000
C00876=88.681,9.321,28.348,-177.1552,-33.9223,0.0000
C00877=89.020,4.801,28.341,-177.8282,-34.0669,0.0000
C00878=89.153,0.000,28.346,180.0000,-34.0969,0.0000
C00879=89.020,-4.801,28.341,177.8282,-34.0669,0.0000
C00880=88.681,-9.321,28.348,177.1552,-33.9223,0.0000
C00881=88.468,-13.530,28.499,-177.7865,-32.1731,0.0000
C00882=88.922,-16.227,28.874,-168.9410,-21.6868,0.0000
C00883=89.999,-18.049,29.382,-171.2088,-9.4842,0.0000
C00884=91.502,-19.567,29.895,-175.9610,-3.5233,0.0000
C00885=93.139,-21.117,30.283,-178.7276,-1.3354,0.0000
C00886=94.499,-23.038,30.474,-179.6218,-0.8308,0.0000
C00887=95.229,-25.943,30.574,-179.9828,-0.1432,0.0000
C00888=95.186,-29.476,30.656,-179.9370,0.4927,0.0000
C00889=94.318,-33.085,30.738,179.9943,-0.0172,0.0000
C00890=93.071,-36.560,30.793,180.0000,-0.0000,0.0000
C00891=91.663,-39.959,30.793,180.0000,-0.0000,0.0000
C00892=90.088,-43.298,30.738,179.9943,-0.0115,0.0000
C00893=88.150,-46.464,30.656,-179.6963,0.3896,0.0000
C00894=85.682,-48.993,30.574,179.8854,-0.0917,0.0000
C00895=83.111,-50.531,30.474,179.1463,-0.3209,0.0000
C00896=80.791,-50.927,30.283,178.1605,-0.0459,0.0000
C00897=78.538,-50.865,29.895,174.6634,0.3626,0.0000
C00898=76.401,-50.876,29.382,167.1853,-0.5053,0.0000
C00899=74.351,-51.403,28.874,157.2499,-8.1354,0.0000
C00900=72.123,-52.989,28.499,154.7223,-22.6602,0.0000
C00901=69.298,-56.115,28.348,156.2276,-27.0522,0.0000
C00902=66.342,-59.552,28.341,155.7090,-26.7916,0.0000
C00903=63.040,-63.040,28.346,154.4202,-25.5798,0.0000
C00904=59.552,-66.342,28.341,153.2084,-24.2910,0.0000
C00905=56.115,-69.298,28.348,152.9478,-23.7724,0.0000
C00906=52.989,-72.123,28.499,157.3398,-25.2777,0.0000
C00907=51.403,-74.351,28.874,171.8646,-22.7501,0.0000
C00908=50.876,-76.401,29.382,179.4947,-12.8147,0.0000
C00909=50.865,-78.538,29.895,-179.6374,-5.3366,0.0000
C00910=50.927,-80.791,30.283,179.9541,-1.8395,0.0000
C00911=50.531,-83.111,30.474,179.6791,-0.8537,0.0000
C00912=48.993,-85.682,30.574,179.9083,-0.1146,0.0000
C00913=46.464,-88.150,30.656,-179.6104,0.3037,0.0000
C00914=43.298,-90.088,30.738,179.9885,-0.0057,0.0000
C00915=39.959,-91.663,30.793,180.0000,-0.0000,0.0000
C00916=36.560,-93.071,30.793,180.0000,-0.0000,0.0000
C00917=33.085,-94.318,30.738,179.9828,-0.0057,0.0000
C00918=29.476,-95.186,30.656,-179.5073,0.0630,0.0000
C00919=25.943,-95.229,30.574,179.8568,0.0172,0.0000
C00920=23.038,-94.499,30.474,179.1692,0.3782,0.0000
C00921=21.117,-93.139,30.283,178.6646,1.2724,0.0000
C00922=19.567,-91.502,29.895,176.4767,4.0390,0.0000
C00923=18.049,-89.999,29.382,170.5158,8.7912,0.0000
C00924=16.227,-88.922,28.874,158.3132,11.0590,0.0000
C00925=13.530,-88.468,28.499,147.8269,2.2135,0.0000
C00926=9.321,-88.681,28.348,146.0777,-2.8448,0.0000
C00927=4.801,-89.020,28.341,145.9331,-2.1718,0.0000
C00928=0.000,-89.153,28.346,145.9031,0.0000,0.0000
C00929=0.000,-89.153,28.346,145.9031,0.0000,0.0000
C00930=-4.801,-89.020,28.341,145.9331,2.1718,0.0000
C00931=-9.321,-88.681,28.348,146.0777,2.8448,0.0000
C00932=-13.530,-88.468,28.499,147.8269,-2.2135,0.0000
C00933=-16.227,-88.922,28.874,158.3132,-11.0590,0.0000
C00934=-18.049,-89.999,29.382,170.5158,-8.7912,0.0000
C00935=-19.567,-91.502,29.895,176.4767,-4.0390,0.0000
C00936=-21.117,-93.139,30.283,178.6646,-1.2724,0.0000
C00937=-23.038,-94.499,30.474,179.1692,-0.3782,0.0000
C00938=-25.943,-95.229,30.574,179.8568,-0.0172,0.0000
C00939=-29.476,-95.186,30.656,-179.5073,-0.0630,0.0000
C00940=-33.085,-94.318,30.738,179.9828,0.0057,0.0000
C00941=-36.560,-93.071,30.793,180.0000,0.0000,0.0000
C00942=-39.959,-91.663,30.793,180.0000,0.0000,0.0000
C00943=-43.298,-90.088,30.738,179.9885,0.0057,0.0000
C00944=-46.464,-88.150,30.656,-179.6104,-0.3037,0.0000
C00945=-48.993,-85.682,30.574,179.9083,0.1146,0.0000
C00946=-50.531,-83.111,30.474,179.6791,0.8537,0.0000
C00947=-50.927,-80.791,30.283,179.9541,1.8395,0.0000
C00948=-50.865,-78.538,29.895,-179.6374,5.3366,0.0000
C00949=-50.876,-76.401,29.382,179.4947,12.8147,0.0000
C00950=-51.403,-74.351,28.874,171.8646,22.7501,0.0000
C00951=-52.989,-72.123,28.499,157.3398,25.2777,0.0000
C00952=-56.115,-69.298,28.348,152.9478,23.7724,0.0000
C00953=-59.552,-66.342,28.341,153.2084,24.2910,0.0000
C00954=-63.040,-63.040,28.346,154.4202,25.5798,0.0000
C00955=-66.342,-59.552,28.341,155.7090,26.7916,0.0000
C00956=-69.298,-56.115,28.348,156.2276,27.0522,0.0000
C00957=-72.123,-52.989,28.499,154.7223,22.6602,0.0000
C00958=-74.351,-51.403,28.874,157.2499,8.1354,0.0000
C00959=-76.401,-50.876,29.382,167.1853,0.5053,0.0000
C00960=-78.538,-50.865,29.895,174.6634,-0.3626,0.0000
C00961=-80.791,-50.927,30.283,178.1605,0.0459,0.0000
C00962=-83.111,-50.531,30.474,179.1463,0.3209,0.0000
C00963=-85.682,-48.993,30.574,179.8854,0.0917,0.0000
C00964=-88.150,-46.464,30.656,-179.6963,-0.3896,0.0000
C00965=-90.088,-43.298,30.738,179.9943,0.0115,0.0000
C00966=-91.663,-39.959,30.793,180.0000,0.0000,0.0000
C00967=-93.071,-36.560,30.793,180.0000,0.0000,0.0000
C00968=-94.318,-33.085,30.738,179.9943,0.0172,0.0000
C00969=-95.186,-29.476,30.656,-179.9370,-0.4927,0.0000
C00970=-95.229,-25.943,30.574,-179.9828,0.1432,0.0000
C00971=-94.499,-23.038,30.474,-179.6218,0.8308,0.0000
C00972=-93.139,-21.117,30.283,-178.7276,1.3354,0.0000
C00973=-91.502,-19.567,29.895,-175.9610,3.5233,0.0000
C00974=-89.999,-18.049,29.382,-171.2088,9.4842,0.0000
C00975=-88.922,-16.227,28.874,-168.9410,21.6868,0.0000
C00976=-88.468,-13.530,28.499,-177.7865,32.1731,0.0000
C00977=-88.681,-9.321,28.348,177.1552,33.9223,0.0000
C00978=-89.020,-4.801,28.341,177.8282,34.0669,0.0000
C00979=-89.153,0.000,28.346,-180.0000,34.0969,0.0000
C00980=-89.020,4.801,28.341,-177.8282,34.0669,0.0000
C00981=-88.681,9.321,28.348,-177.1552,33.9223,0.0000
C00982=-88.468,13.530,28.499,177.7865,32.1731,0.0000
C00983=-88.922,16.227,28.874,168.9410,21.6868,0.0000
C00984=-89.999,18.049,29.382,171.2088,9.4842,0.0000
C00985=-91.502,19.567,29.895,175.9610,3.5233,0.0000
C00986=-93.139,21.117,30.283,178.7276,1.3354,0.0000
C00987=-94.499,23.038,30.474,179.6218,0.8308,0.0000
C00988=-95.229,25.943,30.574,179.9828,0.1432,0.0000
C00989=-95.186,29.476,30.656,179.9370,-0.4927,0.0000
C00990=-94.318,33.085,30.738,-179.9943,0.0172,0.0000
C00991=-93.071,36.560,30.793,-180.0000,0.0000,0.0000
C00992=-91.663,39.959,30.793,-180.0000,0.0000,0.0000
C00993=-90.088,43.298,30.738,-179.9943,0.0115,0.0000
C00994=-88.150,46.464,30.656,179.6963,-0.3896,0.0000
C00995=-85.682,48.993,30.574,-179.8854,0.0917,0.0000
C00996=-83.111,50.531,30.474,-179.1463,0.3209,0.0000
C00997=-80.791,50.927,30.283,-178.1605,0.0459,0.0000
C00998=-78.538,50.865,29.895,-174.6634,-0.3626,0.0000
C00999=-76.401,50.876,29.382,-167.1853,0.5053,0.0000
C01000=-74.351,51.403,28.874,-157.2499,8.1354,0.0000
C01001=-72.123,52.989,28.499,-154.7223,22.6602,0.0000
C01002=-69.298,56.115,28.348,-156.2276,27.0522,0.0000
C01003=-66.342,59.552,28.341,-155.7090,26.7916,0.0000
C01004=-63.040,63.040,28.346,-154.4202,25.5798,0.0000
C01005=-59.552,66.342,28.341,-153.2084,24.2910,0.0000
C01006=-56.115,69.298,28.348,-152.9478,23.7724,0.0000
C01007=-52.989,72.123,28.499,-157.3398,25.2777,0.0000
C01008=-51.403,74.351,28.874,-171.8646,22.7501,0.0000
C01009=-50.876,76.401,29.382,-179.4947,12.8147,0.0000
C01010=-50.865,78.538,29.895,179.6374,5.3366,0.0000
C01011=-50.927,80.791,30.283,-179.9541,1.8395,0.0000
C01012=-50.531,83.111,30.474,-179.6791,0.8537,0.0000
C01013=-48.993,85.682,30.574,-179.9083,0.1146,0.0000
C01014=-46.464,88.150,30.656,179.6104,-0.3037,0.0000
C01015=-43.298,90.088,30.738,-179.9885,0.0057,0.0000
C01016=-39.959,91.663,30.793,-180.0000,0.0000,0.0000
C01017=-36.560,93.071,30.793,-180.0000,0.0000,0.0000
C01018=-33.085,94.318,30.738,-179.9828,0.0057,0.0000
C01019=-29.476,95.186,30.656,179.5073,-0.0630,0.0000
C01020=-25.943,95.229,30.574,-179.8568,-0.0172,0.0000
C01021=-23.038,94.499,30.474,-179.1692,-0.3782,0.0000
C01022=-21.117,93.139,30.283,-178.6646,-1.2724,0.0000
C01023=-19.567,91.502,29.895,-176.4767,-4.0390,0.0000
C01024=-18.049,89.999,29.382,-170.5158,-8.7912,0.0000
C01025=-16.227,88.922,28.874,-158.3132,-11.0590,0.0000
C01026=-13.530,88.468,28.499,-147.8269,-2.2135,0.0000
C01027=-9.321,88.681,28.348,-146.0777,2.8448,0.0000
C01028=-4.801,89.020,28.341,-145.9331,2.1718,0.0000
C01029=0.000,89.153,28.346,-145.9031,0.0000,0.0000
C01030=0.000,87.904,30.157,-144.9432,0.0000,0.0000
C01031=4.687,87.776,30.152,-144.9728,-2.2459,0.0000
C01032=9.129,87.447,30.160,-145.1203,-2.7589,0.0000
C01033=13.294,87.274,30.332,-147.1500,3.3012,0.0000
C01034=15.938,87.830,30.762,-159.7286,12.2335,0.0000
C01035=17.714,89.068,31.347,-172.2294,8.3664,0.0000
C01036=19.200,90.783,31.942,-177.6293,3.1499,0.0000
C01037=20.718,92.664,32.394,-179.6448,0.4011,0.0000
C01038=22.602,94.262,32.617,179.9312,-0.0401,0.0000
C01039=25.531,95.180,32.735,179.6791,-0.0458,0.0000
C01040=29.149,95.246,32.831,179.3181,0.0688,0.0000
C01041=32.878,94.386,32.928,180.0000,0.0000,0.0000
C01042=36.490,93.098,32.991,180.0000,0.0000,0.0000
C01043=40.028,91.633,32.991,180.0000,0.0000,0.0000
C01044=43.493,89.989,32.928,180.0000,0.0000,0.0000
C01045=46.737,87.960,32.831,179.4671,0.4355,0.0000
C01046=49.249,85.356,32.735,179.8109,0.2578,0.0000
C01047=50.671,82.635,32.617,179.9771,0.0745,0.0000
C01048=50.874,80.174,32.394,179.9714,-0.5328,0.0000
C01049=50.617,77.770,31.942,179.4487,-3.8995,0.0000
C01050=50.455,75.506,31.347,179.5676,-11.3380,0.0000
C01051=50.836,73.375,30.762,-173.8466,-22.5136,0.0000
C01052=52.312,71.113,30.332,-157.4223,-26.4475,0.0000
C01053=55.379,68.290,30.160,-152.2098,-24.6527,0.0000
C01054=58.753,65.381,30.152,-152.3781,-25.0763,0.0000
C01055=62.157,62.157,30.157,-153.6144,-26.3912,0.0000
C01056=65.381,58.753,30.152,-154.9237,-27.6219,0.0000
C01057=68.290,55.379,30.160,-155.3473,-27.7848,0.0000
C01058=71.113,52.312,30.332,-153.5580,-22.5777,0.0000
C01059=73.375,50.836,30.762,-157.4864,-6.1534,0.0000
C01060=75.506,50.455,31.347,-168.6620,0.4324,0.0000
C01061=77.770,50.617,31.942,-176.1005,0.5513,0.0000
C01062=80.174,50.874,32.394,-179.4672,0.0286,0.0000
C01063=82.635,50.671,32.617,179.9255,0.0229,0.0000
C01064=85.356,49.249,32.735,179.7422,0.1891,0.0000
C01065=87.960,46.737,32.831,179.5645,0.5329,0.0000
C01066=89.989,43.493,32.928,180.0000,0.0000,0.0000
C01067=91.633,40.028,32.991,180.0000,0.0000,0.0000
C01068=93.098,36.490,32.991,180.0000,0.0000,0.0000
C01069=94.386,32.878,32.928,180.0000,0.0000,0.0000
C01070=95.246,29.149,32.831,179.9312,0.6819,0.0000
C01071=95.180,25.531,32.735,-179.9542,0.3209,0.0000
C01072=94.262,22.602,32.617,-179.9599,0.0688,0.0000
C01073=92.664,20.718,32.394,179.5989,-0.3552,0.0000
C01074=90.783,19.200,31.942,176.8501,-2.3707,0.0000
C01075=89.068,17.714,31.347,171.6336,-7.7706,0.0000
C01076=87.830,15.938,30.762,167.7665,-20.2714,0.0000
C01077=87.274,13.294,30.332,176.6988,-32.8500,0.0000
C01078=87.447,9.129,30.160,-177.2411,-34.8797,0.0000
C01079=87.776,4.687,30.152,-177.7541,-35.0272,0.0000
C01080=87.904,0.000,30.157,180.0000,-35.0568,0.0000
C01081=87.776,-4.687,30.152,177.7611,-35.0272,0.0000
C01082=87.447,-9.130,30.160,177.2481,-34.8797,0.0000
C01083=87.274,-13.294,30.332,-176.6988,-32.8500,0.0000
C01084=87.830,-15.938,30.762,-167.7665,-20.2714,0.0000
C01085=89.068,-17.714,31.347,-171.6336,-7.7706,0.0000
C01086=90.783,-19.200,31.942,-176.8501,-2.3707,0.0000
C01087=92.664,-20.718,32.394,-179.5989,-0.3552,0.0000
C01088=94.262,-22.602,32.617,179.9599,0.0688,0.0000
C01089=95.180,-25.531,32.735,179.9542,0.3209,0.0000
C01090=95.246,-29.149,32.831,-179.9312,0.6819,0.0000
C01091=94.386,-32.878,32.928,-180.0000,0.0000,0.0000
C01092=93.098,-36.490,32.991,-180.0000,0.0000,0.0000
C01093=91.633,-40.028,32.991,-180.0000,0.0000,0.0000
C01094=89.989,-43.493,32.928,-180.0000,0.0000,0.0000
C01095=87.960,-46.737,32.831,-179.5645,0.5329,0.0000
C01096=85.356,-49.249,32.735,-179.7422,0.1891,0.0000
C01097=82.635,-50.671,32.617,-179.9255,0.0229,0.0000
C01098=80.174,-50.874,32.394,179.4672,0.0286,0.0000
C01099=77.770,-50.617,31.942,176.1005,0.5513,0.0000
C01100=75.506,-50.455,31.347,168.6620,0.4324,0.0000
C01101=73.375,-50.836,30.762,157.4864,-6.1534,0.0000
C01102=71.113,-52.312,30.332,153.5525,-22.5777,0.0000
C01103=68.290,-55.379,30.160,155.3473,-27.7902,0.0000
C01104=65.381,-58.753,30.152,154.9237,-27.6219,0.0000
C01105=62.157,-62.157,30.157,153.6088,-26.3856,0.0000
C01106=58.753,-65.381,30.152,152.3781,-25.0763,0.0000
C01107=55.379,-68.290,30.160,152.2152,-24.6527,0.0000
C01108=52.312,-71.113,30.332,157.4223,-26.4420,0.0000
C01109=50.836,-73.375,30.762,173.8466,-22.5136,0.0000
C01110=50.455,-75.506,31.347,-179.5676,-11.3380,0.0000
C01111=50.617,-77.770,31.942,-179.4487,-3.8995,0.0000
C01112=50.874,-80.174,32.394,-179.9714,-0.5328,0.0000
C01113=50.671,-82.635,32.617,-179.9771,0.0745,0.0000
C01114=49.249,-85.356,32.735,-179.8109,0.2578,0.0000
C01115=46.737,-87.960,32.831,-179.4671,0.4355,0.0000
C01116=43.493,-89.989,32.928,-180.0000,0.0000,0.0000
C01117=40.028,-91.633,32.991,-180.0000,0.0000,0.0000
C01118=36.490,-93.098,32.991,-180.0000,0.0000,0.0000
C01119=32.878,-94.386,32.928,-180.0000,0.0000,0.0000
C01120=29.149,-95.246,32.831,-179.3181,0.0688,0.0000
C01121=25.531,-95.180,32.735,-179.6791,-0.0458,0.0000
C01122=22.602,-94.262,32.617,-179.9312,-0.0401,0.0000
C01123=20.718,-92.664,32.394,179.6448,0.4011,0.0000
C01124=19.200,-90.783,31.942,177.6293,3.1499,0.0000
C01125=17.714,-89.068,31.347,172.2294,8.3664,0.0000
C01126=15.938,-87.830,30.762,159.7286,12.2335,0.0000
C01127=13.294,-87.274,30.332,147.1500,3.3012,0.0000
C01128=9.129,-87.447,30.160,145.1203,-2.7589,0.0000
C01129=4.687,-87.776,30.152,144.9728,-2.2459,0.0000
C01130=0.000,-87.904,30.157,144.9432,0.0000,0.0000
C01131=0.000,-87.904,30.157,144.9432,0.0000,0.0000
C01132=-4.687,-87.776,30.152,144.9728,2.2389,0.0000
C01133=-9.130,-87.447,30.160,145.1203,2.7519,0.0000
C01134=-13.294,-87.274,30.332,147.1500,-3.3012,0.0000
C01135=-15.938,-87.830,30.762,159.7286,-12.2335,0.0000
C01136=-17.714,-89.068,31.347,172.2294,-8.3664,0.0000
C01137=-19.200,-90.783,31.942,177.6293,-3.1499,0.0000
C01138=-20.718,-92.664,32.394,179.6448,-0.4011,0.0000
C01139=-22.602,-94.262,32.617,-179.9312,0.0401,0.0000
C01140=-25.531,-95.180,32.735,-179.6791,0.0458,0.0000
C01141=-29.149,-95.246,32.831,-179.3181,-0.0688,0.0000
C01142=-32.878,-94.386,32.928,-180.0000,-0.0000,0.0000
C01143=-36.490,-93.098,32.991,-180.0000,-0.0000,0.0000
C01144=-40.028,-91.633,32.991,-180.0000,-0.0000,0.0000
C01145=-43.493,-89.989,32.928,-180.0000,-0.0000,0.0000
C01146=-46.737,-87.960,32.831,-179.4671,-0.4355,0.0000
C01147=-49.249,-85.356,32.735,-179.8109,-0.2578,0.0000
C01148=-50.671,-82.635,32.617,-179.9771,-0.0745,0.0000
C01149=-50.874,-80.174,32.394,-179.9714,0.5328,0.0000
C01150=-50.617,-77.770,31.942,-179.4487,3.8995,0.0000
C01151=-50.455,-75.506,31.347,-179.5676,11.3380,0.0000
C01152=-50.836,-73.375,30.762,173.8466,22.5136,0.0000
C01153=-52.312,-71.113,30.332,157.4223,26.4475,0.0000
C01154=-55.379,-68.290,30.160,152.2098,24.6527,0.0000
C01155=-58.753,-65.381,30.152,152.3781,25.0763,0.0000
C01156=-62.157,-62.157,30.157,153.6144,26.3912,0.0000
C01157=-65.381,-58.753,30.152,154.9237,27.6219,0.0000
C01158=-68.290,-55.379,30.160,155.3473,27.7848,0.0000
C01159=-71.113,-52.312,30.332,153.5580,22.5777,0.0000
C01160=-73.375,-50.836,30.762,157.4864,6.1534,0.0000
C01161=-75.506,-50.455,31.347,168.6620,-0.4324,0.0000
C01162=-77.770,-50.617,31.942,176.1005,-0.5513,0.0000
C01163=-80.174,-50.874,32.394,179.4672,-0.0286,0.0000
C01164=-82.635,-50.671,32.617,-179.9255,-0.0229,0.0000
C01165=-85.356,-49.249,32.735,-179.7422,-0.1891,0.0000
C01166=-87.960,-46.737,32.831,-179.5645,-0.5329,0.0000
C01167=-89.989,-43.493,32.928,-180.0000,-0.0000,0.0000
C01168=-91.633,-40.028,32.991,-180.0000,-0.0000,0.0000
C01169=-93.098,-36.490,32.991,-180.0000,-0.0000,0.0000
C01170=-94.386,-32.878,32.928,-180.0000,-0.0000,0.0000
C01171=-95.246,-29.149,32.831,-179.9312,-0.6819,0.0000
C01172=-95.180,-25.531,32.735,179.9542,-0.3209,0.0000
C01173=-94.262,-22.602,32.617,179.9599,-0.0688,0.0000
C01174=-92.664,-20.718,32.394,-179.5989,0.3552,0.0000
C01175=-90.783,-19.200,31.942,-176.8501,2.3707,0.0000
C01176=-89.068,-17.714,31.347,-171.6336,7.7706,0.0000
C01177=-87.830,-15.938,30.762,-167.7665,20.2714,0.0000
C01178=-87.274,-13.294,30.332,-176.6988,32.8500,0.0000
C01179=-87.447,-9.129,30.160,177.2411,34.8797,0.0000
C01180=-87.776,-4.687,30.152,177.7541,35.0272,0.0000
C01181=-87.904,0.000,30.157,-180.0000,35.0568,0.0000
C01182=-87.776,4.687,30.152,-177.7611,35.0272,0.0000
C01183=-87.447,9.130,30.160,-177.2481,34.8797,0.0000
C01184=-87.274,13.294,30.332,176.6988,32.8500,0.0000
C01185=-87.830,15.938,30.762,167.7665,20.2714,0.0000
C01186=-89.068,17.714,31.347,171.6336,7.7706,0.0000
C01187=-90.783,19.200,31.942,176.8501,2.3707,0.0000
C01188=-92.664,20.718,32.394,179.5989,0.3552,0.0000
C01189=-94.262,22.602,32.617,-179.9599,-0.0688,0.0000
C01190=-95.180,25.531,32.735,-179.9542,-0.3209,0.0000
C01191=-95.246,29.149,32.831,179.9312,-0.6819,0.0000
C01192=-94.386,32.878,32.928,180.0000,-0.0000,0.0000
C01193=-93.098,36.490,32.991,180.0000,-0.0000,0.0000
C01194=-91.633,40.028,32.991,180.0000,-0.0000,0.0000
C01195=-89.989,43.493,32.928,180.0000,-0.0000,0.0000
C01196=-87.960,46.737,32.831,179.5645,-0.5329,0.0000
C01197=-85.356,49.249,32.735,179.7422,-0.1891,0.0000
C01198=-82.635,50.671,32.617,179.9255,-0.0229,0.0000
C01199=-80.174,50.874,32.394,-179.4672,-0.0286,0.0000
C01200=-77.770,50.617,31.942,-176.1005,-0.5513,0.0000
C01201=-75.506,50.455,31.347,-168.6620,-0.4324,0.0000
C01202=-73.375,50.836,30.762,-157.4864,6.1534,0.0000
C01203=-71.113,52.312,30.332,-153.5525,22.5777,0.0000
C01204=-68.290,55.379,30.160,-155.3473,27.7902,0.0000
C01205=-65.381,58.753,30.152,-154.9237,27.6219,0.0000
C01206=-62.157,62.157,30.157,-153.6088,26.3856,0.0000
C01207=-58.753,65.381,30.152,-152.3781,25.0763,0.0000
C01208=-55.379,68.290,30.160,-152.2152,24.6527,0.0000
C01209=-52.312,71.113,30.332,-157.4223,26.4420,0.0000
C01210=-50.836,73.375,30.762,-173.8466,22.5136,0.0000
C01211=-50.455,75.506,31.347,179.5676,11.3380,0.0000
C01212=-50.617,77.770,31.942,179.4487,3.8995,0.0000
C01213=-50.874,80.174,32.394,179.9714,0.5328,0.0000
C01214=-50.671,82.635,32.617,179.9771,-0.0745,0.0000
C01215=-49.249,85.356,32.735,179.8109,-0.2578,0.0000
C01216=-46.737,87.960,32.831,179.4671,-0.4355,0.0000
C01217=-43.493,89.989,32.928,180.0000,-0.0000,0.0000
C01218=-40.028,91.633,32.991,180.0000,-0.0000,0.0000
C01219=-36.490,93.098,32.991,180.0000,-0.0000,0.0000
C01220=-32.878,94.386,32.928,180.0000,-0.0000,0.0000
C01221=-29.149,95.246,32.831,179.3181,-0.0688,0.0000
C01222=-25.531,95.180,32.735,179.6791,0.0458,0.0000
C01223=-22.602,94.262,32.617,179.9312,0.0401,0.0000
C01224=-20.718,92.664,32.394,-179.6448,-0.4011,0.0000
C01225=-19.200,90.783,31.942,-177.6293,-3.1499,0.0000
C01226=-17.714,89.068,31.347,-172.2294,-8.3664,0.0000
C01227=-15.938,87.830,30.762,-159.7286,-12.2335,0.0000
C01228=-13.294,87.274,30.332,-147.1500,-3.3012,0.0000
C01229=-9.130,87.447,30.160,-145.1203,2.7519,0.0000
C01230=-4.687,87.776,30.152,-144.9728,2.2389,0.0000
C01231=0.000,87.904,30.157,-144.9432,0.0000,0.0000
C01232=0.000,86.627,31.948,-144.1053,0.0000,0.0000
C01233=4.570,86.503,31.943,-144.1345,-2.2977,0.0000
C01234=8.933,86.186,31.951,-144.2837,-2.6320,0.0000
C01235=13.053,86.053,32.146,-146.6507,4.4586,0.0000
C01236=15.641,86.712,32.633,-161.4204,13.0389,0.0000
C01237=17.370,88.113,33.299,-173.7907,7.6704,0.0000
C01238=18.822,90.045,33.980,-178.5722,2.1612,0.0000
C01239=20.308,92.176,34.500,179.5645,-0.5673,0.0000
C01240=22.152,94.017,34.757,179.0889,-0.5960,0.0000
C01241=25.107,95.129,34.893,179.2093,-0.1547,0.0000
C01242=28.812,95.307,35.004,179.1176,0.0745,0.0000
C01243=32.664,94.457,35.116,179.9828,0.0057,0.0000
C01244=36.417,93.126,35.190,179.9943,0.0000,0.0000
C01245=40.099,91.601,35.190,179.9943,0.0000,0.0000
C01246=43.694,89.888,35.116,179.9828,0.0057,0.0000
C01247=47.019,87.765,35.004,179.3239,0.5730,0.0000
C01248=49.513,85.019,34.893,179.5473,0.6704,0.0000
C01249=50.816,82.144,34.757,179.7765,1.0658,0.0000
C01250=50.818,79.538,34.500,-179.9083,0.7105,0.0000
C01251=50.362,76.980,33.980,179.4781,-2.5391,0.0000
C01252=50.022,74.588,33.299,178.9534,-9.7723,0.0000
C01253=50.255,72.374,32.633,-175.7745,-21.8750,0.0000
C01254=51.619,70.079,32.146,-157.6932,-27.4976,0.0000
C01255=54.626,67.259,31.951,-151.5903,-25.4472,0.0000
C01256=57.935,64.399,31.943,-151.6474,-25.7731,0.0000
C01257=61.254,61.254,31.948,-152.8971,-27.1029,0.0000
C01258=64.398,57.936,31.943,-154.2269,-28.3526,0.0000
C01259=67.259,54.626,31.951,-154.5528,-28.4097,0.0000
C01260=70.079,51.619,32.146,-152.5024,-22.3068,0.0000
C01261=72.374,50.255,32.633,-158.1250,-4.2255,0.0000
C01262=74.588,50.022,33.299,-170.2277,1.0466,0.0000
C01263=76.980,50.362,33.980,-177.4609,0.5219,0.0000
C01264=79.538,50.818,34.500,179.2895,-0.0917,0.0000
C01265=82.144,50.816,34.757,178.9342,0.2235,0.0000
C01266=85.019,49.513,34.893,179.3296,0.4527,0.0000
C01267=87.765,47.019,35.004,179.4270,0.6761,0.0000
C01268=89.888,43.694,35.116,179.9943,0.0172,0.0000
C01269=91.601,40.099,35.190,180.0000,0.0057,0.0000
C01270=93.126,36.417,35.190,180.0000,0.0057,0.0000
C01271=94.457,32.664,35.116,179.9943,0.0172,0.0000
C01272=95.307,28.812,35.004,179.9255,0.8824,0.0000
C01273=95.129,25.107,34.893,-179.8453,0.7907,0.0000
C01274=94.017,22.152,34.757,-179.4040,0.9111,0.0000
C01275=92.176,20.308,34.500,-179.4327,0.4355,0.0000
C01276=90.045,18.822,33.980,177.8388,-1.4278,0.0000
C01277=88.113,17.370,33.299,172.3296,-6.2093,0.0000
C01278=86.712,15.641,32.633,166.9611,-18.5796,0.0000
C01279=86.053,13.053,32.146,175.5414,-33.3493,0.0000
C01280=86.186,8.933,31.951,-177.3680,-35.7163,0.0000
C01281=86.503,4.570,31.943,-177.7023,-35.8655,0.0000
C01282=86.627,0.000,31.948,180.0000,-35.8947,0.0000
C01283=86.503,-4.570,31.943,177.7023,-35.8655,0.0000
C01284=86.186,-8.933,31.951,177.3680,-35.7163,0.0000
C01285=86.053,-13.053,32.146,-175.5414,-33.3493,0.0000
C01286=86.712,-15.641,32.633,-166.9611,-18.5796,0.0000
C01287=88.113,-17.370,33.299,-172.3296,-6.2093,0.0000
C01288=90.045,-18.822,33.980,-177.8388,-1.4278,0.0000
C01289=92.176,-20.308,34.500,179.4327,0.4355,0.0000
C01290=94.017,-22.152,34.757,179.4040,0.9111,0.0000
C01291=95.129,-25.107,34.893,179.8453,0.7907,0.0000
C01292=95.307,-28.812,35.004,-179.9255,0.8824,0.0000
C01293=94.457,-32.664,35.116,-179.9943,0.0172,0.0000
C01294=93.126,-36.417,35.190,-180.0000,0.0057,0.0000
C01295=91.601,-40.099,35.190,-180.0000,0.0057,0.0000
C01296=89.888,-43.694,35.116,-179.9943,0.0172,0.0000
C01297=87.765,-47.019,35.004,-179.4270,0.6761,0.0000
C01298=85.019,-49.513,34.893,-179.3296,0.4527,0.0000
C01299=82.144,-50.816,34.757,-178.9342,0.2235,0.0000
C01300=79.538,-50.818,34.500,-179.2895,-0.0917,0.0000
C01301=76.980,-50.362,33.980,177.4609,0.5219,0.0000
C01302=74.588,-50.022,33.299,170.2277,1.0466,0.0000
C01303=72.374,-50.255,32.633,158.1250,-4.2255,0.0000
C01304=70.079,-51.619,32.146,152.5024,-22.3068,0.0000
C01305=67.259,-54.626,31.951,154.5528,-28.4097,0.0000
C01306=64.399,-57.935,31.943,154.2269,-28.3526,0.0000
C01307=61.254,-61.254,31.948,152.8971,-27.1029,0.0000
C01308=57.936,-64.398,31.943,151.6474,-25.7731,0.0000
C01309=54.626,-67.259,31.951,151.5903,-25.4472,0.0000
C01310=51.619,-70.079,32.146,157.6932,-27.4976,0.0000
C01311=50.255,-72.374,32.633,175.7745,-21.8750,0.0000
C01312=50.022,-74.588,33.299,-178.9534,-9.7723,0.0000
C01313=50.362,-76.980,33.980,-179.4781,-2.5391,0.0000
C01314=50.818,-79.538,34.500,179.9083,0.7105,0.0000
C01315=50.816,-82.144,34.757,-179.7765,1.0658,0.0000
C01316=49.513,-85.019,34.893,-179.5473,0.6704,0.0000
C01317=47.019,-87.765,35.004,-179.3239,0.5730,0.0000
C01318=43.694,-89.888,35.116,-179.9828,0.0057,0.0000
C01319=40.099,-91.601,35.190,-179.9943,0.0000,0.0000
C01320=36.417,-93.126,35.190,-179.9943,0.0000,0.0000
C01321=32.664,-94.457,35.116,-179.9828,0.0057,0.0000
C01322=28.812,-95.307,35.004,-179.1176,0.0745,0.0000
C01323=25.107,-95.129,34.893,-179.2093,-0.1547,0.0000
C01324=22.152,-94.017,34.757,-179.0889,-0.5960,0.0000
C01325=20.308,-92.176,34.500,-179.5645,-0.5673,0.0000
C01326=18.822,-90.045,33.980,178.5722,2.1612,0.0000
C01327=17.370,-88.113,33.299,173.7907,7.6704,0.0000
C01328=15.641,-86.712,32.633,161.4204,13.0389,0.0000
C01329=13.053,-86.053,32.146,146.6507,4.4586,0.0000
C01330=8.933,-86.186,31.951,144.2837,-2.6320,0.0000
C01331=4.570,-86.503,31.943,144.1345,-2.2977,0.0000
C01332=0.000,-86.627,31.948,144.1053,0.0000,0.0000
C01333=0.000,-86.627,31.948,144.1053,0.0000,0.0000
C01334=-4.570,-86.503,31.943,144.1345,2.2977,0.0000
C01335=-8.933,-86.186,31.951,144.2837,2.6320,0.0000
C01336=-13.053,-86.053,32.146,146.6507,-4.4586,0.0000
C01337=-15.641,-86.712,32.633,161.4204,-13.0389,0.0000
C01338=-17.370,-88.113,33.299,173.7907,-7.6704,0.0000
C01339=-18.822,-90.045,33.980,178.5722,-2.1612,0.0000
C01340=-20.308,-92.176,34.500,-179.5645,0.5673,0.0000
C01341=-22.152,-94.017,34.757,-179.0889,0.5960,0.0000
C01342=-25.107,-95.129,34.893,-179.2093,0.1547,0.0000
C01343=-28.812,-95.307,35.004,-179.1176,-0.0745,0.0000
C01344=-32.664,-94.457,35.116,-179.9828,-0.0057,0.0000
C01345=-36.417,-93.126,35.190,-179.9943,-0.0000,0.0000
C01346=-40.099,-91.601,35.190,-179.9943,-0.0000,0.0000
C01347=-43.694,-89.888,35.116,-179.9828,-0.0057,0.0000
C01348=-47.019,-87.765,35.004,-179.3239,-0.5730,0.0000
C01349=-49.513,-85.019,34.893,-179.5473,-0.6704,0.0000
C01350=-50.816,-82.144,34.757,-179.7765,-1.0658,0.0000
C01351=-50.818,-79.538,34.500,179.9083,-0.7105,0.0000
C01352=-50.362,-76.980,33.980,-179.4781,2.5391,0.0000
C01353=-50.022,-74.588,33.299,-178.9534,9.7723,0.0000
C01354=-50.255,-72.374,32.633,175.7745,21.8750,0.0000
C01355=-51.619,-70.079,32.146,157.6932,27.4976,0.0000
C01356=-54.626,-67.259,31.951,151.5903,25.4472,0.0000
C01357=-57.935,-64.399,31.943,151.6474,25.7731,0.0000
C01358=-61.254,-61.254,31.948,152.8971,27.1029,0.0000
C01359=-64.398,-57.936,31.943,154.2269,28.3526,0.0000
C01360=-67.259,-54.626,31.951,154.5528,28.4097,0.0000
C01361=-70.079,-51.619,32.146,152.5024,22.3068,0.0000
C01362=-72.374,-50.255,32.633,158.1250,4.2255,0.0000
C01363=-74.588,-50.022,33.299,170.2277,-1.0466,0.0000
C01364=-76.980,-50.362,33.980,177.4609,-0.5219,0.0000
C01365=-79.538,-50.818,34.500,-179.2895,0.0917,0.0000
C01366=-82.144,-50.816,34.757,-178.9342,-0.2235,0.0000
C01367=-85.019,-49.513,34.893,-179.3296,-0.4527,0.0000
C01368=-87.765,-47.019,35.004,-179.4270,-0.6761,0.0000
C01369=-89.888,-43.694,35.116,-179.9943,-0.0172,0.0000
C01370=-91.601,-40.099,35.190,-180.0000,-0.0057,0.0000
C01371=-93.126,-36.417,35.190,-180.0000,-0.0057,0.0000
C01372=-94.457,-32.664,35.116,-179.9943,-0.0172,0.0000
C01373=-95.307,-28.812,35.004,-179.9255,-0.8824,0.0000
C01374=-95.129,-25.107,34.893,179.8453,-0.7907,0.0000
C01375=-94.017,-22.152,34.757,179.4040,-0.9111,0.0000
C01376=-92.176,-20.308,34.500,179.4327,-0.4355,0.0000
C01377=-90.045,-18.822,33.980,-177.8388,1.4278,0.0000
C01378=-88.113,-17.370,33.299,-172.3296,6.2093,0.0000
C01379=-86.712,-15.641,32.633,-166.9611,18.5796,0.0000
C01380=-86.053,-13.053,32.146,-175.5414,33.3493,0.0000
C01381=-86.186,-8.933,31.951,177.3680,35.7163,0.0000
C01382=-86.503,-4.570,31.943,177.7023,35.8655,0.0000
C01383=-86.627,0.000,31.948,-180.0000,35.8947,0.0000
C01384=-86.503,4.570,31.943,-177.7023,35.8655,0.0000
C01385=-86.186,8.933,31.951,-177.3680,35.7163,0.0000
C01386=-86.053,13.053,32.146,175.5414,33.3493,0.0000
C01387=-86.712,15.641,32.633,166.9611,18.5796,0.0000
C01388=-88.113,17.370,33.299,172.3296,6.2093,0.0000
C01389=-90.045,18.822,33.980,177.8388,1.4278,0.0000
C01390=-92.176,20.308,34.500,-179.4327,-0.4355,0.0000
C01391=-94.017,22.152,34.757,-179.4040,-0.9111,0.0000
C01392=-95.129,25.107,34.893,-179.8453,-0.7907,0.0000
C01393=-95.307,28.812,35.004,179.9255,-0.8824,0.0000
C01394=-94.457,32.664,35.116,179.9943,-0.0172,0.0000
C01395=-93.126,36.417,35.190,180.0000,-0.0057,0.0000
C01396=-91.601,40.099,35.190,180.0000,-0.0057,0.0000
C01397=-89.888,43.694,35.116,179.9943,-0.0172,0.0000
C01398=-87.765,47.019,35.004,179.4270,-0.6761,0.0000
C01399=-85.019,49.513,34.893,179.3296,-0.4527,0.0000
C01400=-82.144,50.816,34.757,178.9342,-0.2235,0.0000
C01401=-79.538,50.818,34.500,179.2895,0.0917,0.0000
C01402=-76.980,50.362,33.980,-177.4609,-0.5219,0.0000
C01403=-74.588,50.022,33.299,-170.2277,-1.0466,0.0000
C01404=-72.374,50.255,32.633,-158.1250,4.2255,0.0000
C01405=-70.079,51.619,32.146,-152.5024,22.3068,0.0000
C01406=-67.259,54.626,31.951,-154.5528,28.4097,0.0000
C01407=-64.399,57.935,31.943,-154.2269,28.3526,0.0000
C01408=-61.254,61.254,31.948,-152.8971,27.1029,0.0000
C01409=-57.936,64.398,31.943,-151.6474,25.7731,0.0000
C01410=-54.626,67.259,31.951,-151.5903,25.4472,0.0000
C01411=-51.619,70.079,32.146,-157.6932,27.4976,0.0000
C01412=-50.255,72.374,32.633,-175.7745,21.8750,0.0000
C01413=-50.022,74.588,33.299,178.9534,9.7723,0.0000
C01414=-50.362,76.980,33.980,179.4781,2.5391,0.0000
C01415=-50.818,79.538,34.500,-179.9083,-0.7105,0.0000
C01416=-50.816,82.144,34.757,179.7765,-1.0658,0.0000
C01417=-49.513,85.019,34.893,179.5473,-0.6704,0.0000
C01418=-47.019,87.765,35.004,179.3239,-0.5730,0.0000
C01419=-43.694,89.888,35.116,179.9828,-0.0057,0.0000
C01420=-40.099,91.601,35.190,179.9943,-0.0000,0.0000
C01421=-36.417,93.126,35.190,179.9943,-0.0000,0.0000
C01422=-32.664,94.457,35.116,179.9828,-0.0057,0.0000
C01423=-28.812,95.307,35.004,179.1176,-0.0745,0.0000
C01424=-25.107,95.129,34.893,179.2093,0.1547,0.0000
C01425=-22.152,94.017,34.757,179.0889,0.5960,0.0000
C01426=-20.308,92.176,34.500,179.5645,0.5673,0.0000
C01427=-18.822,90.045,33.980,-178.5722,-2.1612,0.0000
C01428=-17.370,88.113,33.299,-173.7907,-7.6704,0.0000
C01429=-15.641,86.712,32.633,-161.4204,-13.0389,0.0000
C01430=-13.053,86.053,32.146,-146.6507,-4.4586,0.0000
C01431=-8.933,86.186,31.951,-144.2837,2.6320,0.0000
C01432=-4.570,86.503,31.943,-144.1345,2.2977,0.0000
C01433=0.000,86.627,31.948,-144.1053,0.0000,0.0000
C01434=0.000,85.325,33.722,-143.3719,0.0000,0.0000
C01435=4.451,85.206,33.716,-143.4007,-2.3479,0.0000
C01436=8.733,84.900,33.725,-143.5612,-2.4855,0.0000
C01437=12.808,84.808,33.943,-146.3179,5.6607,0.0000
C01438=15.338,85.570,34.490,-163.2996,13.4572,0.0000
C01439=17.019,87.137,35.239,-175.1592,6.7891,0.0000
C01440=18.435,89.289,36.009,-179.3295,1.1518,0.0000
C01441=19.887,91.675,36.600,178.9453,-1.5588,0.0000
C01442=21.692,93.766,36.894,178.3320,-1.2555,0.0000
C01443=24.671,95.076,37.049,178.7336,-0.2980,0.0000
C01444=28.465,95.370,37.176,178.9228,0.0688,0.0000
C01445=32.445,94.529,37.304,179.9656,0.0115,0.0000
C01446=36.342,93.155,37.389,179.9943,0.0000,0.0000
C01447=40.172,91.569,37.389,179.9943,0.0000,0.0000
C01448=43.901,89.784,37.304,179.9714,0.0172,0.0000
C01449=47.309,87.565,37.176,179.1863,0.7106,0.0000
C01450=49.784,84.674,37.049,179.3180,1.1060,0.0000
C01451=50.965,81.641,36.894,179.7076,2.0689,0.0000
C01452=50.762,78.886,36.600,-179.6446,1.8452,0.0000
C01453=50.101,76.172,36.009,179.6619,-1.2893,0.0000
C01454=49.580,73.649,35.239,178.6106,-8.2006,0.0000
C01455=49.662,71.353,34.490,-177.5405,-20.8782,0.0000
C01456=50.912,69.025,33.943,-158.1402,-28.4267,0.0000
C01457=53.858,66.209,33.725,-151.0690,-26.1703,0.0000
C01458=57.102,63.397,33.716,-151.0097,-26.3877,0.0000
C01459=60.334,60.334,33.722,-152.2677,-27.7323,0.0000
C01460=63.397,57.102,33.716,-153.6123,-28.9903,0.0000
C01461=66.209,53.858,33.725,-153.8297,-28.9310,0.0000
C01462=69.025,50.912,33.943,-151.5733,-21.8598,0.0000
C01463=71.353,49.662,34.490,-159.1218,-2.4595,0.0000
C01464=73.649,49.580,35.239,-171.7994,1.3894,0.0000
C01465=76.172,50.101,36.009,-178.7107,0.3381,0.0000
C01466=78.886,50.762,36.600,178.1548,-0.3554,0.0000
C01467=81.641,50.965,36.894,177.9311,0.2924,0.0000
C01468=84.674,49.784,37.049,178.8940,0.6820,0.0000
C01469=87.565,47.309,37.176,179.2894,0.8137,0.0000
C01470=89.784,43.901,37.304,179.9828,0.0286,0.0000
C01471=91.569,40.172,37.389,180.0000,0.0057,0.0000
C01472=93.155,36.342,37.389,180.0000,0.0057,0.0000
C01473=94.529,32.445,37.304,179.9885,0.0344,0.0000
C01474=95.370,28.465,37.176,179.9312,1.0772,0.0000
C01475=95.076,24.671,37.049,-179.7020,1.2664,0.0000
C01476=93.766,21.692,36.894,-178.7445,1.6680,0.0000
C01477=91.675,19.887,36.600,-178.4412,1.0547,0.0000
C01478=89.289,18.435,36.009,178.8482,-0.6705,0.0000
C01479=87.137,17.019,35.239,173.2109,-4.8408,0.0000
C01480=85.570,15.338,34.490,166.5428,-16.7004,0.0000
C01481=84.808,12.808,33.943,174.3393,-33.6821,0.0000
C01482=84.900,8.733,33.725,-177.5145,-36.4388,0.0000
C01483=85.206,4.451,33.716,-177.6521,-36.5993,0.0000
C01484=85.325,0.000,33.722,180.0000,-36.6281,0.0000
C01485=85.206,-4.451,33.716,177.6521,-36.5993,0.0000
C01486=84.900,-8.733,33.725,177.5145,-36.4388,0.0000
C01487=84.808,-12.808,33.943,-174.3462,-33.6821,0.0000
C01488=85.570,-15.338,34.490,-166.5428,-16.7004,0.0000
C01489=87.137,-17.019,35.239,-173.2109,-4.8408,0.0000
C01490=89.289,-18.435,36.009,-178.8482,-0.6705,0.0000
C01491=91.675,-19.887,36.600,178.4412,1.0547,0.0000
C01492=93.766,-21.692,36.894,178.7445,1.6680,0.0000
C01493=95.076,-24.671,37.049,179.7020,1.2664,0.0000
C01494=95.370,-28.465,37.176,-179.9312,1.0772,0.0000
C01495=94.529,-32.445,37.304,-179.9885,0.0344,0.0000
C01496=93.155,-36.342,37.389,-180.0000,0.0057,0.0000
C01497=91.569,-40.172,37.389,-180.0000,0.0057,0.0000
C01498=89.784,-43.901,37.304,-179.9828,0.0286,0.0000
C01499=87.565,-47.309,37.176,-179.2894,0.8137,0.0000
C01500=84.674,-49.784,37.049,-178.8940,0.6820,0.0000
C01501=81.641,-50.965,36.894,-177.9311,0.2924,0.0000
C01502=78.886,-50.762,36.600,-178.1548,-0.3554,0.0000
C01503=76.172,-50.101,36.009,178.7107,0.3381,0.0000
C01504=73.649,-49.580,35.239,171.7994,1.3894,0.0000
C01505=71.353,-49.662,34.490,159.1218,-2.4595,0.0000
C01506=69.025,-50.912,33.943,151.5733,-21.8598,0.0000
C01507=66.209,-53.858,33.725,153.8297,-28.9310,0.0000
C01508=63.397,-57.102,33.716,153.6123,-28.9903,0.0000
C01509=60.334,-60.334,33.722,152.2677,-27.7323,0.0000
C01510=57.102,-63.397,33.716,151.0097,-26.3877,0.0000
C01511=53.858,-66.209,33.725,151.0690,-26.1703,0.0000
C01512=50.912,-69.025,33.943,158.1402,-28.4267,0.0000
C01513=49.662,-71.353,34.490,177.5405,-20.8782,0.0000
C01514=49.580,-73.649,35.239,-178.6106,-8.2006,0.0000
C01515=50.101,-76.172,36.009,-179.6619,-1.2893,0.0000
C01516=50.762,-78.886,36.600,179.6446,1.8452,0.0000
C01517=50.965,-81.641,36.894,-179.7076,2.0689,0.0000
C01518=49.784,-84.674,37.049,-179.3180,1.1060,0.0000
C01519=47.309,-87.565,37.176,-179.1863,0.7106,0.0000
C01520=43.901,-89.784,37.304,-179.9714,0.0172,0.0000
C01521=40.172,-91.569,37.389,-179.9943,0.0000,0.0000
C01522=36.342,-93.155,37.389,-179.9943,0.0000,0.0000
C01523=32.445,-94.529,37.304,-179.9656,0.0115,0.0000
C01524=28.465,-95.370,37.176,-178.9228,0.0688,0.0000
C01525=24.671,-95.076,37.049,-178.7336,-0.2980,0.0000
C01526=21.692,-93.766,36.894,-178.3320,-1.2555,0.0000
C01527=19.887,-91.675,36.600,-178.9453,-1.5588,0.0000
C01528=18.435,-89.289,36.009,179.3295,1.1518,0.0000
C01529=17.019,-87.137,35.239,175.1592,6.7891,0.0000
C01530=15.338,-85.570,34.490,163.2996,13.4572,0.0000
C01531=12.808,-84.808,33.943,146.3179,5.6607,0.0000
C01532=8.733,-84.900,33.725,143.5612,-2.4855,0.0000
C01533=4.451,-85.206,33.716,143.4007,-2.3479,0.0000
C01534=0.000,-85.325,33.722,143.3719,0.0000,0.0000
C01535=0.000,-85.325,33.722,143.3719,0.0000,0.0000
C01536=-4.451,-85.206,33.716,143.4007,2.3479,0.0000
C01537=-8.733,-84.900,33.725,143.5612,2.4855,0.0000
C01538=-12.808,-84.808,33.943,146.3179,-5.6538,0.0000
C01539=-15.338,-85.570,34.490,163.2996,-13.4572,0.0000
C01540=-17.019,-87.137,35.239,175.1592,-6.7891,0.0000
C01541=-18.435,-89.289,36.009,179.3295,-1.1518,0.0000
C01542=-19.887,-91.675,36.600,-178.9453,1.5588,0.0000
C01543=-21.692,-93.766,36.894,-178.3320,1.2555,0.0000
C01544=-24.671,-95.076,37.049,-178.7336,0.2980,0.0000
C01545=-28.465,-95.370,37.176,-178.9228,-0.0688,0.0000
C01546=-32.445,-94.529,37.304,-179.9656,-0.0115,0.0000
C01547=-36.342,-93.155,37.389,-179.9943,-0.0000,0.0000
C01548=-40.172,-91.569,37.389,-179.9943,-0.0000,0.0000
C01549=-43.901,-89.784,37.304,-179.9714,-0.0172,0.0000
C01550=-47.309,-87.565,37.176,-179.1863,-0.7106,0.0000
C01551=-49.784,-84.674,37.049,-179.3180,-1.1060,0.0000
C01552=-50.965,-81.641,36.894,-179.7076,-2.0689,0.0000
C01553=-50.762,-78.886,36.600,179.6446,-1.8452,0.0000
C01554=-50.101,-76.172,36.009,-179.6619,1.2893,0.0000
C01555=-49.580,-73.649,35.239,-178.6106,8.2006,0.0000
C01556=-49.662,-71.353,34.490,177.5405,20.8782,0.0000
C01557=-50.912,-69.025,33.943,158.1402,28.4267,0.0000
C01558=-53.858,-66.209,33.725,151.0690,26.1703,0.0000
C01559=-57.102,-63.397,33.716,151.0097,26.3877,0.0000
C01560=-60.334,-60.334,33.722,152.2677,27.7323,0.0000
C01561=-63.397,-57.102,33.716,153.6123,28.9903,0.0000
C01562=-66.209,-53.858,33.725,153.8297,28.9310,0.0000
C01563=-69.025,-50.912,33.943,151.5733,21.8598,0.0000
C01564=-71.353,-49.662,34.490,159.1218,2.4595,0.0000
C01565=-73.649,-49.580,35.239,171.7994,-1.3894,0.0000
C01566=-76.172,-50.101,36.009,178.7107,-0.3381,0.0000
C01567=-78.886,-50.762,36.600,-178.1548,0.3554,0.0000
C01568=-81.641,-50.965,36.894,-177.9311,-0.2924,0.0000
C01569=-84.674,-49.784,37.049,-178.8940,-0.6820,0.0000
C01570=-87.565,-47.309,37.176,-179.2894,-0.8137,0.0000
C01571=-89.784,-43.901,37.304,-179.9828,-0.0286,0.0000
C01572=-91.569,-40.172,37.389,-180.0000,-0.0057,0.0000
C01573=-93.155,-36.342,37.389,-180.0000,-0.0057,0.0000
C01574=-94.529,-32.445,37.304,-179.9885,-0.0344,0.0000
C01575=-95.370,-28.465,37.176,-179.9312,-1.0772,0.0000
C01576=-95.076,-24.671,37.049,179.7020,-1.2664,0.0000
C01577=-93.766,-21.692,36.894,178.7445,-1.6680,0.0000
C01578=-91.675,-19.887,36.600,178.4412,-1.0547,0.0000
C01579=-89.289,-18.435,36.009,-178.8482,0.6705,0.0000
C01580=-87.137,-17.019,35.239,-173.2109,4.8408,0.0000
C01581=-85.570,-15.338,34.490,-166.5428,16.7004,0.0000
C01582=-84.808,-12.808,33.943,-174.3393,33.6821,0.0000
C01583=-84.900,-8.733,33.725,177.5145,36.4388,0.0000
C01584=-85.206,-4.451,33.716,177.6521,36.5993,0.0000
C01585=-85.325,0.000,33.722,-180.0000,36.6281,0.0000
C01586=-85.206,4.451,33.716,-177.6521,36.5993,0.0000
C01587=-84.900,8.733,33.725,-177.5145,36.4388,0.0000
C01588=-84.808,12.808,33.943,174.3462,33.6821,0.0000
C01589=-85.570,15.338,34.490,166.5428,16.7004,0.0000
C01590=-87.137,17.019,35.239,173.2109,4.8408,0.0000
C01591=-89.289,18.435,36.009,178.8482,0.6705,0.0000
C01592=-91.675,19.887,36.600,-178.4412,-1.0547,0.0000
C01593=-93.766,21.692,36.894,-178.7445,-1.6680,0.0000
C01594=-95.076,24.671,37.049,-179.7020,-1.2664,0.0000
C01595=-95.370,28.465,37.176,179.9312,-1.0772,0.0000
C01596=-94.529,32.445,37.304,179.9885,-0.0344,0.0000
C01597=-93.155,36.342,37.389,180.0000,-0.0057,0.0000
C01598=-91.569,40.172,37.389,180.0000,-0.0057,0.0000
C01599=-89.784,43.901,37.304,179.9828,-0.0286,0.0000
C01600=-87.565,47.309,37.176,179.2894,-0.8137,0.0000
C01601=-84.674,49.784,37.049,178.8940,-0.6820,0.0000
C01602=-81.641,50.965,36.894,177.9311,-0.2924,0.0000
C01603=-78.886,50.762,36.600,178.1548,0.3554,0.0000
C01604=-76.172,50.101,36.009,-178.7107,-0.3381,0.0000
C01605=-73.649,49.580,35.239,-171.7994,-1.3894,0.0000
C01606=-71.353,49.662,34.490,-159.1218,2.4595,0.0000
C01607=-69.025,50.912,33.943,-151.5733,21.8598,0.0000
C01608=-66.209,53.858,33.725,-153.8297,28.9310,0.0000
C01609=-63.397,57.102,33.716,-153.6123,28.9903,0.0000
C01610=-60.334,60.334,33.722,-152.2677,27.7323,0.0000
C01611=-57.102,63.397,33.716,-151.0097,26.3877,0.0000
C01612=-53.858,66.209,33.725,-151.0690,26.1703,0.0000
C01613=-50.912,69.025,33.943,-158.1402,28.4267,0.0000
C01614=-49.662,71.353,34.490,-177.5405,20.8782,0.0000
C01615=-49.580,73.649,35.239,178.6106,8.2006,0.0000
C01616=-50.101,76.172,36.009,179.6619,1.2893,0.0000
C01617=-50.762,78.886,36.600,-179.6446,-1.8452,0.0000
C01618=-50.965,81.641,36.894,179.7076,-2.0689,0.0000
C01619=-49.784,84.674,37.049,179.3180,-1.1060,0.0000
C01620=-47.309,87.565,37.176,179.1863,-0.7106,0.0000
C01621=-43.901,89.784,37.304,179.9714,-0.0172,0.0000
C01622=-40.172,91.569,37.389,179.9943,-0.0000,0.0000
C01623=-36.342,93.155,37.389,179.9943,-0.0000,0.0000
C01624=-32.445,94.529,37.304,179.9656,-0.0115,0.0000
C01625=-28.465,95.370,37.176,178.9228,-0.0688,0.0000
C01626=-24.671,95.076,37.049,178.7336,0.2980,0.0000
C01627=-21.692,93.766,36.894,178.3320,1.2555,0.0000
C01628=-19.887,91.675,36.600,178.9453,1.5588,0.0000
C01629=-18.435,89.289,36.009,-179.3295,-1.1518,0.0000
C01630=-17.019,87.137,35.239,-175.1592,-6.7891,0.0000
C01631=-15.338,85.570,34.490,-163.2996,-13.4572,0.0000
C01632=-12.808,84.808,33.943,-146.3179,-5.6538,0.0000
C01633=-8.733,84.900,33.725,-143.5612,2.4855,0.0000
C01634=-4.451,85.206,33.716,-143.4007,2.3479,0.0000
C01635=0.000,85.325,33.722,-143.3719,0.0000,0.0000
C01636=0.000,84.003,35.480,-142.7416,0.0000,0.0000
C01637=4.330,83.888,35.473,-142.7701,-2.3889,0.0000
C01638=8.530,83.594,35.484,-142.9375,-2.3047,0.0000
C01639=12.558,83.543,35.726,-146.1534,6.8791,0.0000
C01640=15.030,84.409,36.333,-165.2561,13.5084,0.0000
C01641=16.662,86.143,37.169,-176.3234,5.7969,0.0000
C01642=18.041,88.518,38.031,-179.9198,0.1547,0.0000
C01643=19.458,91.164,38.697,178.4915,-2.5227,0.0000
C01644=21.221,93.510,39.027,177.6890,-1.9844,0.0000
C01645=24.227,95.023,39.203,178.2751,-0.4758,0.0000
C01646=28.112,95.435,39.346,178.7280,0.0573,0.0000
C01647=32.220,94.603,39.491,179.9542,0.0172,0.0000
C01648=36.266,93.184,39.587,179.9943,0.0000,0.0000
C01649=40.247,91.535,39.587,179.9943,0.0057,0.0000
C01650=44.111,89.678,39.491,179.9542,0.0229,0.0000
C01651=47.604,87.360,39.346,179.0602,0.8595,0.0000
C01652=50.060,84.322,39.203,179.1173,1.5531,0.0000
C01653=51.116,81.128,39.027,179.7705,3.0324,0.0000
C01654=50.704,78.221,38.697,-179.2829,2.8490,0.0000
C01655=49.835,75.348,38.031,179.9484,-0.1662,0.0000
C01656=49.130,72.694,37.169,178.4885,-6.6864,0.0000
C01657=49.058,70.314,36.333,-179.0756,-19.5929,0.0000
C01658=50.194,67.954,35.726,-158.7482,-29.2286,0.0000
C01659=53.078,65.141,35.484,-150.6450,-26.8231,0.0000
C01660=56.256,62.380,35.473,-150.4587,-26.9210,0.0000
C01661=59.399,59.399,35.480,-151.7250,-28.2750,0.0000
C01662=62.380,56.256,35.473,-153.0790,-29.5413,0.0000
C01663=65.141,53.078,35.484,-153.1769,-29.3550,0.0000
C01664=67.954,50.194,35.726,-150.7714,-21.2518,0.0000
C01665=70.314,49.058,36.333,-160.4071,-0.9244,0.0000
C01666=72.694,49.130,37.169,-173.3136,1.5115,0.0000
C01667=75.348,49.835,38.031,-179.8338,0.0516,0.0000
C01668=78.221,50.704,38.697,177.1510,-0.7171,0.0000
C01669=81.128,51.116,39.027,176.9676,0.2295,0.0000
C01670=84.322,50.060,39.203,178.4469,0.8827,0.0000
C01671=87.360,47.604,39.346,179.1405,0.9398,0.0000
C01672=89.678,44.111,39.491,179.9771,0.0458,0.0000
C01673=91.535,40.247,39.587,179.9943,0.0057,0.0000
C01674=93.184,36.266,39.587,180.0000,0.0057,0.0000
C01675=94.603,32.220,39.491,179.9828,0.0458,0.0000
C01676=95.435,28.112,39.346,179.9427,1.2720,0.0000
C01677=95.023,24.227,39.203,-179.5242,1.7249,0.0000
C01678=93.510,21.221,39.027,-178.0156,2.3110,0.0000
C01679=91.164,19.458,38.697,-177.4773,1.5085,0.0000
C01680=88.518,18.041,38.031,179.8453,-0.0802,0.0000
C01681=86.143,16.662,37.169,174.2031,-3.6766,0.0000
C01682=84.409,15.030,36.333,166.4916,-14.7439,0.0000
C01683=83.543,12.558,35.726,173.1209,-33.8466,0.0000
C01684=83.594,8.530,35.484,-177.6953,-37.0625,0.0000
C01685=83.888,4.330,35.473,-177.6111,-37.2299,0.0000
C01686=84.003,0.000,35.480,180.0000,-37.2584,0.0000
C01687=83.888,-4.330,35.473,177.6111,-37.2299,0.0000
C01688=83.594,-8.530,35.484,177.7025,-37.0625,0.0000
C01689=83.543,-12.558,35.726,-173.1209,-33.8466,0.0000
C01690=84.409,-15.030,36.333,-166.4916,-14.7439,0.0000
C01691=86.143,-16.662,37.169,-174.2031,-3.6766,0.0000
C01692=88.518,-18.041,38.031,-179.8453,-0.0802,0.0000
C01693=91.164,-19.458,38.697,177.4773,1.5085,0.0000
C01694=93.510,-21.221,39.027,178.0156,2.3110,0.0000
C01695=95.023,-24.227,39.203,179.5242,1.7249,0.0000
C01696=95.435,-28.112,39.346,-179.9427,1.2720,0.0000
C01697=94.603,-32.220,39.491,-179.9828,0.0458,0.0000
C01698=93.184,-36.266,39.587,-180.0000,0.0057,0.0000
C01699=91.535,-40.247,39.587,-179.9943,0.0057,0.0000
C01700=89.678,-44.111,39.491,-179.9771,0.0458,0.0000
C01701=87.360,-47.604,39.346,-179.1405,0.9398,0.0000
C01702=84.322,-50.060,39.203,-178.4469,0.8827,0.0000
C01703=81.128,-51.116,39.027,-176.9676,0.2295,0.0000
C01704=78.221,-50.704,38.697,-177.1510,-0.7171,0.0000
C01705=75.348,-49.835,38.031,179.8338,0.0516,0.0000
C01706=72.694,-49.130,37.169,173.3136,1.5115,0.0000
C01707=70.314,-49.058,36.333,160.4071,-0.9244,0.0000
C01708=67.954,-50.194,35.726,150.7714,-21.2518,0.0000
C01709=65.141,-53.078,35.484,153.1769,-29.3550,0.0000
C01710=62.380,-56.256,35.473,153.0790,-29.5413,0.0000
C01711=59.399,-59.399,35.480,151.7250,-28.2750,0.0000
C01712=56.256,-62.380,35.473,150.4587,-26.9210,0.0000
C01713=53.078,-65.141,35.484,150.6450,-26.8231,0.0000
C01714=50.194,-67.954,35.726,158.7482,-29.2286,0.0000
C01715=49.058,-70.314,36.333,179.0756,-19.5929,0.0000
C01716=49.130,-72.694,37.169,-178.4885,-6.6864,0.0000
C01717=49.835,-75.348,38.031,-179.9484,-0.1662,0.0000
C01718=50.704,-78.221,38.697,179.2829,2.8490,0.0000
C01719=51.116,-81.128,39.027,-179.7705,3.0324,0.0000
C01720=50.060,-84.322,39.203,-179.1173,1.5531,0.0000
C01721=47.604,-87.360,39.346,-179.0602,0.8595,0.0000
C01722=44.111,-89.678,39.491,-179.9542,0.0229,0.0000
C01723=40.247,-91.535,39.587,-179.9943,0.0057,0.0000
C01724=36.266,-93.184,39.587,-179.9943,0.0000,0.0000
C01725=32.220,-94.603,39.491,-179.9542,0.0172,0.0000
C01726=28.112,-95.435,39.346,-178.7280,0.0573,0.0000
C01727=24.227,-95.023,39.203,-178.2751,-0.4758,0.0000
C01728=21.221,-93.510,39.027,-177.6890,-1.9844,0.0000
C01729=19.458,-91.164,38.697,-178.4915,-2.5227,0.0000
C01730=18.041,-88.518,38.031,179.9198,0.1547,0.0000
C01731=16.662,-86.143,37.169,176.3234,5.7969,0.0000
C01732=15.030,-84.409,36.333,165.2561,13.5084,0.0000
C01733=12.558,-83.543,35.726,146.1534,6.8791,0.0000
C01734=8.530,-83.594,35.484,142.9375,-2.3047,0.0000
C01735=4.330,-83.888,35.473,142.7701,-2.3889,0.0000
C01736=0.000,-84.003,35.480,142.7416,0.0000,0.0000
C01737=0.000,-84.003,35.480,142.7416,0.0000,0.0000
C01738=-4.330,-83.888,35.473,142.7701,2.3889,0.0000
C01739=-8.530,-83.594,35.484,142.9375,2.2975,0.0000
C01740=-12.558,-83.543,35.726,146.1534,-6.8791,0.0000
C01741=-15.030,-84.409,36.333,165.2561,-13.5084,0.0000
C01742=-16.662,-86.143,37.169,176.3234,-5.7969,0.0000
C01743=-18.041,-88.518,38.031,179.9198,-0.1547,0.0000
C01744=-19.458,-91.164,38.697,-178.4915,2.5227,0.0000
C01745=-21.221,-93.510,39.027,-177.6890,1.9844,0.0000
C01746=-24.227,-95.023,39.203,-178.2751,0.4758,0.0000
C01747=-28.112,-95.435,39.346,-178.7280,-0.0573,0.0000
C01748=-32.220,-94.603,39.491,-179.9542,-0.0172,0.0000
C01749=-36.266,-93.184,39.587,-179.9943,-0.0000,0.0000
C01750=-40.247,-91.535,39.587,-179.9943,-0.0057,0.0000
C01751=-44.111,-89.678,39.491,-179.9542,-0.0229,0.0000
C01752=-47.604,-87.360,39.346,-179.0602,-0.8595,0.0000
C01753=-50.060,-84.322,39.203,-179.1173,-1.5531,0.0000
C01754=-51.116,-81.128,39.027,-179.7705,-3.0324,0.0000
C01755=-50.704,-78.221,38.697,179.2829,-2.8490,0.0000
C01756=-49.835,-75.348,38.031,-179.9484,0.1662,0.0000
C01757=-49.130,-72.694,37.169,-178.4885,6.6864,0.0000
C01758=-49.058,-70.314,36.333,179.0756,19.5929,0.0000
C01759=-50.194,-67.954,35.726,158.7482,29.2286,0.0000
C01760=-53.078,-65.141,35.484,150.6450,26.8231,0.0000
C01761=-56.256,-62.380,35.473,150.4587,26.9210,0.0000
C01762=-59.399,-59.399,35.480,151.7250,28.2750,0.0000
C01763=-62.380,-56.256,35.473,153.0790,29.5413,0.0000
C01764=-65.141,-53.078,35.484,153.1769,29.3550,0.0000
C01765=-67.954,-50.194,35.726,150.7714,21.2518,0.0000
C01766=-70.314,-49.058,36.333,160.4071,0.9244,0.0000
C01767=-72.694,-49.130,37.169,173.3136,-1.5115,0.0000
C01768=-75.348,-49.835,38.031,179.8338,-0.0516,0.0000
C01769=-78.221,-50.704,38.697,-177.1510,0.7171,0.0000
C01770=-81.128,-51.116,39.027,-176.9676,-0.2295,0.0000
C01771=-84.322,-50.060,39.203,-178.4469,-0.8827,0.0000
C01772=-87.360,-47.604,39.346,-179.1405,-0.9398,0.0000
C01773=-89.678,-44.111,39.491,-179.9771,-0.0458,0.0000
C01774=-91.535,-40.247,39.587,-179.9943,-0.0057,0.0000
C01775=-93.184,-36.266,39.587,-180.0000,-0.0057,0.0000
C01776=-94.603,-32.220,39.491,-179.9828,-0.0458,0.0000
C01777=-95.435,-28.112,39.346,-179.9427,-1.2720,0.0000
C01778=-95.023,-24.227,39.203,179.5242,-1.7249,0.0000
C01779=-93.510,-21.221,39.027,178.0156,-2.3110,0.0000
C01780=-91.164,-19.458,38.697,177.4773,-1.5085,0.0000
C01781=-88.518,-18.041,38.031,-179.8453,0.0802,0.0000
C01782=-86.143,-16.662,37.169,-174.2031,3.6766,0.0000
C01783=-84.409,-15.030,36.333,-166.4916,14.7439,0.0000
C01784=-83.543,-12.558,35.726,-173.1209,33.8466,0.0000
C01785=-83.594,-8.530,35.484,177.6953,37.0625,0.0000
C01786=-83.888,-4.330,35.473,177.6111,37.2299,0.0000
C01787=-84.003,0.000,35.480,-180.0000,37.2584,0.0000
C01788=-83.888,4.330,35.473,-177.6111,37.2299,0.0000
C01789=-83.594,8.530,35.484,-177.7025,37.0625,0.0000
C01790=-83.543,12.558,35.726,173.1209,33.8466,0.0000
C01791=-84.409,15.030,36.333,166.4916,14.7439,0.0000
C01792=-86.143,16.662,37.169,174.2031,3.6766,0.0000
C01793=-88.518,18.041,38.031,179.8453,0.0802,0.0000
C01794=-91.164,19.458,38.697,-177.4773,-1.5085,0.0000
C01795=-93.510,21.221,39.027,-178.0156,-2.3110,0.0000
C01796=-95.023,24.227,39.203,-179.5242,-1.7249,0.0000
C01797=-95.435,28.112,39.346,179.9427,-1.2720,0.0000
C01798=-94.603,32.220,39.491,179.9828,-0.0458,0.0000
C01799=-93.184,36.266,39.587,180.0000,-0.0057,0.0000
C01800=-91.535,40.247,39.587,179.9943,-0.0057,0.0000
C01801=-89.678,44.111,39.491,179.9771,-0.0458,0.0000
C01802=-87.360,47.604,39.346,179.1405,-0.9398,0.0000
C01803=-84.322,50.060,39.203,178.4469,-0.8827,0.0000
C01804=-81.128,51.116,39.027,176.9676,-0.2295,0.0000
C01805=-78.221,50.704,38.697,177.1510,0.7171,0.0000
C01806=-75.348,49.835,38.031,-179.8338,-0.0516,0.0000
C01807=-72.694,49.130,37.169,-173.3136,-1.5115,0.0000
C01808=-70.314,49.058,36.333,-160.4071,0.9244,0.0000
C01809=-67.954,50.194,35.726,-150.7714,21.2518,0.0000
C01810=-65.141,53.078,35.484,-153.1769,29.3550,0.0000
C01811=-62.380,56.256,35.473,-153.0790,29.5413,0.0000
C01812=-59.399,59.399,35.480,-151.7250,28.2750,0.0000
C01813=-56.256,62.380,35.473,-150.4587,26.9210,0.0000
C01814=-53.078,65.141,35.484,-150.6450,26.8231,0.0000
C01815=-50.194,67.954,35.726,-158.7482,29.2286,0.0000
C01816=-49.058,70.314,36.333,-179.0756,19.5929,0.0000
C01817=-49.130,72.694,37.169,178.4885,6.6864,0.0000
C01818=-49.835,75.348,38.031,179.9484,0.1662,0.0000
C01819=-50.704,78.221,38.697,-179.2829,-2.8490,0.0000
C01820=-51.116,81.128,39.027,179.7705,-3.0324,0.0000
C01821=-50.060,84.322,39.203,179.1173,-1.5531,0.0000
C01822=-47.604,87.360,39.346,179.0602,-0.8595,0.0000
C01823=-44.111,89.678,39.491,179.9542,-0.0229,0.0000
C01824=-40.247,91.535,39.587,179.9943,-0.0057,0.0000
C01825=-36.266,93.184,39.587,179.9943,-0.0000,0.0000
C01826=-32.220,94.603,39.491,179.9542,-0.0172,0.0000
C01827=-28.112,95.435,39.346,178.7280,-0.0573,0.0000
C01828=-24.227,95.023,39.203,178.2751,0.4758,0.0000
C01829=-21.221,93.510,39.027,177.6890,1.9844,0.0000
C01830=-19.458,91.164,38.697,178.4915,2.5227,0.0000
C01831=-18.041,88.518,38.031,-179.9198,-0.1547,0.0000
C01832=-16.662,86.143,37.169,-176.3234,-5.7969,0.0000
C01833=-15.030,84.409,36.333,-165.2561,-13.5084,0.0000
C01834=-12.558,83.543,35.726,-146.1534,-6.8791,0.0000
C01835=-8.530,83.594,35.484,-142.9375,2.2975,0.0000
C01836=-4.330,83.888,35.473,-142.7701,2.3889,0.0000
C01837=0.000,84.003,35.480,-142.7416,0.0000,0.0000
C01838=0.000,82.662,37.225,-142.2064,0.0000,0.0000
C01839=4.208,82.553,37.217,-142.2346,-2.4206,0.0000
C01840=8.324,82.270,37.229,-142.4136,-2.0895,0.0000
C01841=12.305,82.260,37.495,-146.1467,8.1087,0.0000
C01842=14.718,83.232,38.165,-167.2085,13.2264,0.0000
C01843=16.299,85.134,39.090,-177.2969,4.7546,0.0000
C01844=17.640,87.735,40.048,179.6333,-0.7850,0.0000
C01845=19.021,90.644,40.789,178.1744,-3.4301,0.0000
C01846=20.743,93.250,41.159,177.1708,-2.7375,0.0000
C01847=23.775,94.968,41.355,177.8450,-0.6823,0.0000
C01848=27.752,95.500,41.515,178.5446,0.0401,0.0000
C01849=31.992,94.679,41.678,179.9370,0.0172,0.0000
C01850=36.189,93.214,41.785,179.9943,0.0057,0.0000
C01851=40.323,91.502,41.785,179.9943,0.0057,0.0000
C01852=44.326,89.570,41.678,179.9427,0.0286,0.0000
C01853=47.905,87.153,41.515,178.9398,1.0029,0.0000
C01854=50.341,83.964,41.355,178.9565,2.0061,0.0000
C01855=51.270,80.606,41.159,179.9368,3.9338,0.0000
C01856=50.645,77.545,40.789,-178.8631,3.7161,0.0000
C01857=49.565,74.511,40.048,-179.7020,0.8194,0.0000
C01858=48.673,71.724,39.090,178.5442,-5.2686,0.0000
C01859=48.447,69.261,38.165,179.6745,-18.0961,0.0000
C01860=49.465,66.868,37.495,-159.5148,-29.8988,0.0000
C01861=52.288,64.059,37.229,-150.3112,-27.4065,0.0000
C01862=55.398,61.349,37.217,-149.9872,-27.3801,0.0000
C01863=58.451,58.451,37.225,-151.2622,-28.7378,0.0000
C01864=61.349,55.398,37.217,-152.6199,-30.0128,0.0000
C01865=64.059,52.288,37.229,-152.5935,-29.6888,0.0000
C01866=66.868,49.465,37.495,-150.1012,-20.4913,0.0000
C01867=69.261,48.447,38.165,-161.9039,0.3255,0.0000
C01868=71.724,48.673,39.090,-174.7314,1.4558,0.0000
C01869=74.511,49.565,40.048,179.1806,-0.2980,0.0000
C01870=77.545,50.645,40.789,176.2839,-1.1369,0.0000
C01871=80.606,51.270,41.159,176.0662,0.0632,0.0000
C01872=83.964,50.341,41.355,177.9939,1.0435,0.0000
C01873=87.153,47.905,41.515,178.9971,1.0602,0.0000
